// NETWORK 6
Timer3(
    BOOL_SIGNAL_IN := CollectTimerComplete OR bDirectDrainInProcess,
    BOOL_TIMER_RST := NOT bMainOnOff OR NOT bDirectDrainInProcess,
    INT_AUTO_RST := 1,
    INT_SV_SEC := iDrainingTimer); // DOWN_COUNT_TIMER
DrainComplete := Timer3.SIGNAL_BOOL;

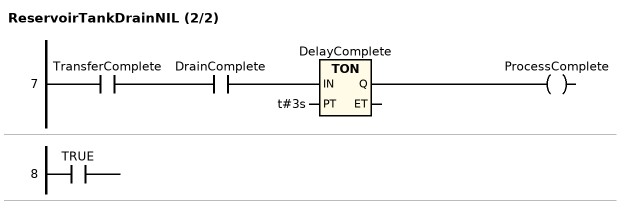
// NETWORK 7
DelayComplete(IN := TransferComplete AND DrainComplete, PT := t#3s); // TON
ProcessComplete := DelayComplete.Q;

// NETWORK 8

END_FUNCTION_BLOCK

// ---- FBs/B_JKS_NewFB/FBP-ArmRelated/fbA1_ArmHorzPosMemory.TcPOU
FUNCTION_BLOCK fbA1_ArmHorzPosMemory

VAR_INPUT PERSISTENT
	DSA1ArmHorzPosInput : DSA1_ArmHorzPosInput;
END_VAR



VAR_OUTPUT PERSISTENT
	DSA1ArmHorzPosOutput : DSA1_ArmHorzPosOutput;
END_VAR


VAR PERSISTENT

	iToleranceP: INT;

	lrBufferLdHookPosToleranceP: LREAL;
	lrBufferLdUnhookPosToleranceP: LREAL;
	lrBufferUldHookPosToleranceP: LREAL;
	lrBufferUldUnhookPosToleranceP: LREAL;

	ARlrBufferStnHookPosToleranceP: ARRAY [0..iHorzArmPosArrayQty] OF LREAL;
	ARlrBufferStnUnhookPosToleranceP: ARRAY [0..iHorzArmPosArrayQty] OF LREAL;

	iToleranceN: INT;

	lrBufferLdHookPosToleranceN: LREAL;
	lrBufferLdUnhookPosToleranceN: LREAL;
	lrBufferUldHookPosToleranceN: LREAL;
	lrBufferUldUnhookPosToleranceN: LREAL;

	ARlrBufferStnHookPosToleranceN: ARRAY [0..iHorzArmPosArrayQty] OF LREAL;
	ARlrBufferStnUnhookPosToleranceN: ARRAY [0..iHorzArmPosArrayQty] OF LREAL;

	i2ndSpdP: INT;

	lrBufferLdHookPos2ndSpdP: LREAL;
	lrBufferLdUnhookPos2ndSpdP: LREAL;
	lrBufferUldHookPos2ndSpdP: LREAL;
	lrBufferUldUnhookPos2ndSpdP: LREAL;

	ARlrBufferStnHookPos2ndSpdP: ARRAY [0..iHorzArmPosArrayQty] OF LREAL;
	ARlrBufferStnUnhookPos2ndSpdP: ARRAY [0..iHorzArmPosArrayQty] OF LREAL;

	i2ndSpdN: INT;

	lrBufferLdHookPos2ndSpdN: LREAL;
	lrBufferLdUnhookPos2ndSpdN: LREAL;
	lrBufferUldHookPos2ndSpdN: LREAL;
	lrBufferUldUnhookPos2ndSpdN: LREAL;

	ARlrBufferStnHookPos2ndSpdN: ARRAY [0..iHorzArmPosArrayQty] OF LREAL;
	ARlrBufferStnUnhookPos2ndSpdN: ARRAY [0..iHorzArmPosArrayQty] OF LREAL;
END_VAR

VAR
	iPosConfirmFL: INT;
	i2ndSpdFL: INT;
END_VAR

(* Generate Positive Tolerance *)
(*[][][][][][][][][][][][][][][][][][][][][][][][][][][][][][][][][][][][][][][][][][][][][][][][][][][][][][][][][][][][][][][][][][][][][][][][][][][][][][][][][][][][][][][][][][][][][][][][][][][]*)

lrBufferLdHookPosToleranceP := DSA1ArmHorzPosInput.lrLdHookPos + DSA1ArmHorzPosInput.lrPosConfirmToleranceSV;
lrBufferLdUnhookPosToleranceP := DSA1ArmHorzPosInput.lrLdUnhookPos + DSA1ArmHorzPosInput.lrPosConfirmToleranceSV;
lrBufferUldHookPosToleranceP := DSA1ArmHorzPosInput.lrUldHookPos + DSA1ArmHorzPosInput.lrPosConfirmToleranceSV;
lrBufferUldUnhookPosToleranceP := DSA1ArmHorzPosInput.lrUldUnhookPos + DSA1ArmHorzPosInput.lrPosConfirmToleranceSV;

iToleranceP := 1;

FOR iToleranceP := 1 TO iHorzArmPosArrayQty DO
	ARlrBufferStnHookPosToleranceP[iToleranceP] := DSA1ArmHorzPosInput.ARlrStnHookPos[iToleranceP] + DSA1ArmHorzPosInput.lrPosConfirmToleranceSV;
	ARlrBufferStnUnhookPosToleranceP[iToleranceP] := DSA1ArmHorzPosInput.ARlrStnUnhookPos[iToleranceP] + DSA1ArmHorzPosInput.lrPosConfirmToleranceSV;
END_FOR


(*[][][][][][][][][][][][][][][][][][][][][][][][][][][][][][][][][][][][][][][][][][][][][][][][][][][][][][][][][][][][][][][][][][][][][][][][][][][][][][][][][][][][][][][][][][][][][][][][][][][]*)


(* Generate Negative Tolerance *)
(*[][][][][][][][][][][][][][][][][][][][][][][][][][][][][][][][][][][][][][][][][][][][][][][][][][][][][][][][][][][][][][][][][][][][][][][][][][][][][][][][][][][][][][][][][][][][][][][][][][][]*)

lrBufferLdHookPosToleranceN := DSA1ArmHorzPosInput.lrLdHookPos - DSA1ArmHorzPosInput.lrPosConfirmToleranceSV;
lrBufferLdUnhookPosToleranceN := DSA1ArmHorzPosInput.lrLdUnhookPos - DSA1ArmHorzPosInput.lrPosConfirmToleranceSV;
lrBufferUldHookPosToleranceN := DSA1ArmHorzPosInput.lrUldHookPos - DSA1ArmHorzPosInput.lrPosConfirmToleranceSV;
lrBufferUldUnhookPosToleranceN := DSA1ArmHorzPosInput.lrUldUnhookPos - DSA1ArmHorzPosInput.lrPosConfirmToleranceSV;

iToleranceN := 1;

FOR iToleranceN := 1 TO iHorzArmPosArrayQty DO
	ARlrBufferStnHookPosToleranceN[iToleranceN] := DSA1ArmHorzPosInput.ARlrStnHookPos[iToleranceN] - DSA1ArmHorzPosInput.lrPosConfirmToleranceSV;
	ARlrBufferStnUnhookPosToleranceN[iToleranceN] := DSA1ArmHorzPosInput.ARlrStnUnhookPos[iToleranceN] - DSA1ArmHorzPosInput.lrPosConfirmToleranceSV;
END_FOR


(*[][][][][][][][][][][][][][][][][][][][][][][][][][][][][][][][][][][][][][][][][][][][][][][][][][][][][][][][][][][][][][][][][][][][][][][][][][][][][][][][][][][][][][][][][][][][][][][][][][][]*)



(* Generate Positive 2ndSpeed *)
(*[][][][][][][][][][][][][][][][][][][][][][][][][][][][][][][][][][][][][][][][][][][][][][][][][][][][][][][][][][][][][][][][][][][][][][][][][][][][][][][][][][][][][][][][][][][][][][][][][][][]*)

lrBufferLdHookPos2ndSpdP := DSA1ArmHorzPosInput.lrLdHookPos + DSA1ArmHorzPosInput.lr2ndSpeedSV;
lrBufferLdUnhookPos2ndSpdP := DSA1ArmHorzPosInput.lrLdUnhookPos + DSA1ArmHorzPosInput.lr2ndSpeedSV;
lrBufferUldHookPos2ndSpdP := DSA1ArmHorzPosInput.lrUldHookPos + DSA1ArmHorzPosInput.lr2ndSpeedSV;
lrBufferUldUnhookPos2ndSpdP := DSA1ArmHorzPosInput.lrUldUnhookPos + DSA1ArmHorzPosInput.lr2ndSpeedSV;

i2ndSpdP := 1;

FOR i2ndSpdP := 1 TO iHorzArmPosArrayQty DO
	ARlrBufferStnHookPos2ndSpdP[i2ndSpdP] := DSA1ArmHorzPosInput.ARlrStnHookPos[i2ndSpdP] + DSA1ArmHorzPosInput.lr2ndSpeedSV;
	ARlrBufferStnUnhookPos2ndSpdP[i2ndSpdP] := DSA1ArmHorzPosInput.ARlrStnUnhookPos[i2ndSpdP] + DSA1ArmHorzPosInput.lr2ndSpeedSV;
END_FOR


(*[][][][][][][][][][][][][][][][][][][][][][][][][][][][][][][][][][][][][][][][][][][][][][][][][][][][][][][][][][][][][][][][][][][][][][][][][][][][][][][][][][][][][][][][][][][][][][][][][][][]*)


(* Generate Negative 2ndSpeed *)
(*[][][][][][][][][][][][][][][][][][][][][][][][][][][][][][][][][][][][][][][][][][][][][][][][][][][][][][][][][][][][][][][][][][][][][][][][][][][][][][][][][][][][][][][][][][][][][][][][][][][]*)

lrBufferLdHookPos2ndSpdN := DSA1ArmHorzPosInput.lrLdHookPos - DSA1ArmHorzPosInput.lr2ndSpeedSV;
lrBufferLdUnhookPos2ndSpdN := DSA1ArmHorzPosInput.lrLdUnhookPos - DSA1ArmHorzPosInput.lr2ndSpeedSV;
lrBufferUldHookPos2ndSpdN := DSA1ArmHorzPosInput.lrUldHookPos - DSA1ArmHorzPosInput.lr2ndSpeedSV;
lrBufferUldUnhookPos2ndSpdN := DSA1ArmHorzPosInput.lrUldUnhookPos - DSA1ArmHorzPosInput.lr2ndSpeedSV;

i2ndSpdN := 1;

FOR i2ndSpdN := 1 TO iHorzArmPosArrayQty DO
	ARlrBufferStnHookPos2ndSpdN[i2ndSpdN] := DSA1ArmHorzPosInput.ARlrStnHookPos[i2ndSpdN] - DSA1ArmHorzPosInput.lr2ndSpeedSV;
	ARlrBufferStnUnhookPos2ndSpdN[i2ndSpdN] := DSA1ArmHorzPosInput.ARlrStnUnhookPos[i2ndSpdN] - DSA1ArmHorzPosInput.lr2ndSpeedSV;
END_FOR


(*[][][][][][][][][][][][][][][][][][][][][][][][][][][][][][][][][][][][][][][][][][][][][][][][][][][][][][][][][][][][][][][][][][][][][][][][][][][][][][][][][][][][][][][][][][][][][][][][][][][]*)


(*Generate Pos Confirm Bit*)
(*[][][][][][][][][][][][][][][][][][][][][][][][][][][][][][][][][][][][][][][][][][][][][][][][][][][][][][][][][][][][][][][][][][][][][][][][][][][][][][][][][][][][][][][][][][][][][][][][][][][]*)
IF DSA1ArmHorzPosInput.lrCurrentPos >= lrBufferLdHookPosToleranceN  AND DSA1ArmHorzPosInput.lrCurrentPos <= lrBufferLdHookPosToleranceP THEN
DSA1ArmHorzPosOutput.bLdHookPosConfirm := TRUE;
ELSE
DSA1ArmHorzPosOutput.bLdHookPosConfirm := FALSE;
END_IF

IF DSA1ArmHorzPosInput.lrCurrentPos >= lrBufferLdUnhookPosToleranceN  AND DSA1ArmHorzPosInput.lrCurrentPos <= lrBufferLdUnhookPosToleranceP THEN
DSA1ArmHorzPosOutput.bLdUnhookPosConfirm := TRUE;
ELSE
DSA1ArmHorzPosOutput.bLdUnhookPosConfirm := FALSE;
END_IF

IF DSA1ArmHorzPosInput.lrCurrentPos >= lrBufferUldHookPosToleranceN  AND DSA1ArmHorzPosInput.lrCurrentPos <= lrBufferUldHookPosToleranceP THEN
DSA1ArmHorzPosOutput.bUldHookPosConfirm := TRUE;
ELSE
DSA1ArmHorzPosOutput.bUldHookPosConfirm := FALSE;
END_IF

IF DSA1ArmHorzPosInput.lrCurrentPos >= lrBufferUldUnhookPosToleranceN  AND DSA1ArmHorzPosInput.lrCurrentPos <= lrBufferUldUnhookPosToleranceP THEN
DSA1ArmHorzPosOutput.bUldUnhookPosConfirm := TRUE;
ELSE
DSA1ArmHorzPosOutput.bUldUnhookPosConfirm := FALSE;
END_IF


iPosConfirmFL := 1;
FOR iPosConfirmFL := 1 TO iHorzArmPosArrayQty DO

		IF DSA1ArmHorzPosInput.lrCurrentPos >= ARlrBufferStnHookPosToleranceN[iPosConfirmFL]  AND DSA1ArmHorzPosInput.lrCurrentPos <= ARlrBufferStnHookPosToleranceP[iPosConfirmFL] THEN
		DSA1ArmHorzPosOutput.ARbStnHookPosConfirm[iPosConfirmFL] := TRUE;
		ELSE
		DSA1ArmHorzPosOutput.ARbStnHookPosConfirm[iPosConfirmFL] := FALSE;
		END_IF

		IF DSA1ArmHorzPosInput.lrCurrentPos >= ARlrBufferStnUnhookPosToleranceN[iPosConfirmFL]  AND DSA1ArmHorzPosInput.lrCurrentPos <= ARlrBufferStnUnhookPosToleranceP[iPosConfirmFL] THEN
		DSA1ArmHorzPosOutput.ARbStnUnhookPosConfirm[iPosConfirmFL] := TRUE;
		ELSE
		DSA1ArmHorzPosOutput.ARbStnUnhookPosConfirm[iPosConfirmFL] := FALSE;
		END_IF

END_FOR

(*[][][][][][][][][][][][][][][][][][][][][][][][][][][][][][][][][][][][][][][][][][][][][][][][][][][][][][][][][][][][][][][][][][][][][][][][][][][][][][][][][][][][][][][][][][][][][][][][][][][]*)



(*Generate 2nd Speed Bit*)
(*[][][][][][][][][][][][][][][][][][][][][][][][][][][][][][][][][][][][][][][][][][][][][][][][][][][][][][][][][][][][][][][][][][][][][][][][][][][][][][][][][][][][][][][][][][][][][][][][][][][]*)
IF DSA1ArmHorzPosInput.lrCurrentPos >= lrBufferLdHookPos2ndSpdN  AND DSA1ArmHorzPosInput.lrCurrentPos <= lrBufferLdHookPos2ndSpdP AND DSA1ArmHorzPosInput.lrTargetPos = DSA1ArmHorzPosInput.lrLdHookPos THEN


DSA1ArmHorzPosOutput.bLdHook2ndSpeedEn := TRUE;
ELSE
DSA1ArmHorzPosOutput.bLdHook2ndSpeedEn := FALSE;
END_IF

IF DSA1ArmHorzPosInput.lrCurrentPos >= lrBufferLdUnhookPos2ndSpdN  AND DSA1ArmHorzPosInput.lrCurrentPos <= lrBufferLdUnhookPos2ndSpdP AND DSA1ArmHorzPosInput.lrTargetPos = DSA1ArmHorzPosInput.lrLdUnhookPos THEN
DSA1ArmHorzPosOutput.bLdUnhook2ndSpeedEn := TRUE;
ELSE
DSA1ArmHorzPosOutput.bLdUnhook2ndSpeedEn := FALSE;
END_IF

IF DSA1ArmHorzPosInput.lrCurrentPos >= lrBufferUldHookPos2ndSpdN  AND DSA1ArmHorzPosInput.lrCurrentPos <= lrBufferUldHookPos2ndSpdP AND DSA1ArmHorzPosInput.lrTargetPos = DSA1ArmHorzPosInput.lrUldHookPos THEN
DSA1ArmHorzPosOutput.bUldHook2ndSpeedEn := TRUE;
ELSE
DSA1ArmHorzPosOutput.bUldHook2ndSpeedEn := FALSE;
END_IF

IF DSA1ArmHorzPosInput.lrCurrentPos >= lrBufferUldUnhookPos2ndSpdN  AND DSA1ArmHorzPosInput.lrCurrentPos <= lrBufferUldUnhookPos2ndSpdP AND DSA1ArmHorzPosInput.lrTargetPos = DSA1ArmHorzPosInput.lrUldUnhookPos THEN
DSA1ArmHorzPosOutput.bUldUnhook2ndSpeedEn := TRUE;
ELSE
DSA1ArmHorzPosOutput.bUldUnhook2ndSpeedEn := FALSE;
END_IF


i2ndSpdFL := 1;
FOR i2ndSpdFL := 1 TO iHorzArmPosArrayQty DO

	IF DSA1ArmHorzPosInput.lrCurrentPos >= ARlrBufferStnHookPos2ndSpdN[i2ndSpdFL]  AND DSA1ArmHorzPosInput.lrCurrentPos <= ARlrBufferStnHookPos2ndSpdP[i2ndSpdFL] AND DSA1ArmHorzPosInput.lrTargetPos = DSA1ArmHorzPosInput.ARlrStnHookPos[i2ndSpdFL] THEN
	DSA1ArmHorzPosOutput.ARbStnHook2ndSpeedEn[i2ndSpdFL] := TRUE;
	ELSE
	DSA1ArmHorzPosOutput.ARbStnHook2ndSpeedEn[i2ndSpdFL] := FALSE;
	END_IF

	IF DSA1ArmHorzPosInput.lrCurrentPos >= ARlrBufferStnUnhookPos2ndSpdN[i2ndSpdFL]  AND DSA1ArmHorzPosInput.lrCurrentPos <= ARlrBufferStnUnhookPos2ndSpdP[i2ndSpdFL] AND DSA1ArmHorzPosInput.lrTargetPos = DSA1ArmHorzPosInput.ARlrStnUnhookPos[i2ndSpdFL] THEN
	DSA1ArmHorzPosOutput.ARbStnUnhook2ndSpeedEn[i2ndSpdFL] := TRUE;
	ELSE
	DSA1ArmHorzPosOutput.ARbStnUnhook2ndSpeedEn[i2ndSpdFL] := FALSE;
	END_IF

END_FOR

(*[][][][][][][][][][][][][][][][][][][][][][][][][][][][][][][][][][][][][][][][][][][][][][][][][][][][][][][][][][][][][][][][][][][][][][][][][][][][][][][][][][][][][][][][][][][][][][][][][][][]*)




(*
IN

	DSA1ArmHorzPosInput.lrTargetPos

	DSA1ArmHorzPosInput.lrPosConfirmToleranceSV
	DSA1ArmHorzPosInput.lr2ndSpeedSV

	DSA1ArmHorzPosInput.lrLdHookPos
	DSA1ArmHorzPosInput.lrLdUnhookPos

	DSA1ArmHorzPosInput.lrUldHookPos 
	DSA1ArmHorzPosInput.lrUldUnhookPos

	DSA1ArmHorzPosInput.ARlrStnHookPos
	DSA1ArmHorzPosInput.ARlrStnUnhookPos


OUT

	DSA1ArmHorzPosOutput.bLdHookPosConfirm
	DSA1ArmHorzPosOutput.bLdUnhookPosConfirm
	DSA1ArmHorzPosOutput.bUldHookPosConfirm
	DSA1ArmHorzPosOutput.bUldUnhookPosConfirm
	DSA1ArmHorzPosOutput.ARbStnHookPosConfirm
	DSA1ArmHorzPosOutput.ARbStnUnhookPosConfirm

	DSA1ArmHorzPosOutput.bLdHook2ndSpeedEn
	DSA1ArmHorzPosOutput.bLdUnhook2ndSpeedEn 
	DSA1ArmHorzPosOutput.bUldHook2ndSpeedEn
	DSA1ArmHorzPosOutput.bUldUnhook2ndSpeedEn 
	DSA1ArmHorzPosOutput.ARbStnHook2ndSpeedEn
	DSA1ArmHorzPosOutput.ARbStnUnhook2ndSpeedEn
*)

END_FUNCTION_BLOCK

// ---- FBs/B_JKS_NewFB/FBP-ArmRelated/fbFBPArmHorzZoneConfirm.TcPOU
FUNCTION_BLOCK fbFBPArmHorzZoneConfirm
VAR_INPUT
	bEnable 					: BOOL;
(*	iLdStnID					: INT;
	iUldStnID					: INT;
*)	lrHorzActualPos 			: LREAL;
	lrHorzStartPoint 			: LREAL;
	lrHorzEndPoint 			: LREAL;
	lrLdHorzCentrePoint 		: LREAL;
	ARlrStnHorzCentrePoint 	: ARRAY [1..iStnQty] OF LREAL;
	lrUldHorzCentrePoint 		: LREAL;
	ARiStnHorzListing 		: ARRAY [1..50] OF INT;

END_VAR


VAR_OUTPUT
	bLdHorzZoneConfirm 		: BOOL;
	ARbHorzStnZoneConfirm 	: ARRAY [1..iStnQty] OF BOOL;
	bUldHorzZoneConfirm 		: BOOL;
	ICurrentHorzZoneNo 			: INT;
	bInvalidListingErr				: BOOL;



END_VAR
(*
VAR_IN_OUT
	iZoneEndPoint : ARRAY [1..20] OF INT;
	iActualPos: INT;

END_VAR
*)
VAR

	iActualPos: INT;


	bEnableRE: R_TRIG;
	iGenZoneFL: INT;
	ARlrZoneCentrePoint : ARRAY [1..50] OF LREAL;
	ARlrZoneEndPoint : ARRAY [1..50] OF LREAL;
	ARbZonePosConfirmInt : ARRAY [1..50] OF BOOL;
	iCheckListFL: INT;
	iEndPointFL: INT;
	bEnableFE: F_TRIG;
	iClearFL: INT;
	IZonePosCfFL: INT;
	iCurrentStnFL: INT;
	bCheckStnConfirm: BOOL;
	iCheckStnBitFL: INT;
END_VAR

(*bEnable Rising Edge*)
bEnableRE(CLK:=bEnable , Q=> );
bEnableFE(CLK:=bEnable , Q=> );

(*Generate Zone Centre Point and Transfer Confirm Bit*)
IF bEnable THEN
iGenZoneFL := 1;
	FOR iGenZoneFL := 1 TO 50 DO
		IF iGenZoneFL >= 1 AND iGenZoneFL <= 50 THEN

			IF ARiStnHorzListing[iGenZoneFL] = iLdStnID THEN
				ARlrZoneCentrePoint[iGenZoneFL] := lrLdHorzCentrePoint;
				bLdHorzZoneConfirm := ARbZonePosConfirmInt[iGenZoneFL];
			END_IF

			IF ARiStnHorzListing[iGenZoneFL] = iUldStnID THEN
				ARlrZoneCentrePoint[iGenZoneFL] := lrUldHorzCentrePoint;
				bUldHorzZoneConfirm := ARbZonePosConfirmInt[iGenZoneFL];
			END_IF

			IF ARiStnHorzListing[iGenZoneFL] <> iUldStnID AND ARiStnHorzListing[iGenZoneFL] <> iUldStnID AND ARiStnHorzListing[iGenZoneFL] <> 0 AND ARiStnHorzListing[iGenZoneFL] <= iStnQty THEN
				ARlrZoneCentrePoint[iGenZoneFL] := ARlrStnHorzCentrePoint[ARiStnHorzListing[iGenZoneFL]];
				ARbHorzStnZoneConfirm[ARiStnHorzListing[iGenZoneFL]] := ARbZonePosConfirmInt[iGenZoneFL];
			END_IF
		END_IF
	END_FOR
END_IF


(*Check invalid Stn Listing*)
IF bEnableRE.Q THEN
bInvalidListingErr := FALSE;
iCheckListFL := 1;
	FOR iCheckListFL := 1 TO 50 DO
		IF iCheckListFL >= 1 AND iCheckListFL <= 50 THEN

			IF iCheckListFL = 1 AND ARlrZoneCentrePoint[1] <= 0 THEN
			bInvalidListingErr := TRUE;
			iCheckListFL := 50+1;
			END_IF

			IF iCheckListFL > 1 AND ARlrZoneCentrePoint[iCheckListFL] <= ARlrZoneCentrePoint[iCheckListFL-1] AND ARiStnHorzListing[iCheckListFL] >0 THEN
			bInvalidListingErr := TRUE;
			iCheckListFL := 50+1;
			END_IF
		END_IF
	END_FOR
END_IF




(*Generate End Point *)
IF bEnableRE.Q THEN
iEndPointFL := 1;
	FOR iEndPointFL := 1 TO 50 DO
		IF iEndPointFL >= 1 AND iEndPointFL <= 50-1 THEN

(*			IF iEndPointFL >1 THEN*)
				IF ((ARlrZoneCentrePoint[iEndPointFL+1] - ARlrZoneCentrePoint[iEndPointFL])/2) >0 THEN
				ARlrZoneEndPoint[iEndPointFL] := ((ARlrZoneCentrePoint[iEndPointFL+1] - ARlrZoneCentrePoint[iEndPointFL])/2)+ARlrZoneCentrePoint[iEndPointFL];
				ELSIF lrHorzEndPoint <= ARlrZoneCentrePoint[iEndPointFL] THEN
				ARlrZoneEndPoint[iEndPointFL] := ARlrZoneCentrePoint[iEndPointFL]+5000;
				iEndPointFL := 50+1;
				ELSIF lrHorzEndPoint > ARlrZoneCentrePoint[iEndPointFL] THEN
				ARlrZoneEndPoint[iEndPointFL] := lrHorzEndPoint+1;
				iEndPointFL := 50+1;
				END_IF
(*			END_IF*)
		END_IF
	END_FOR
END_IF


(*Clear Data*)
IF bEnableFE.Q THEN
iClearFL := 1;
	FOR iClearFL := 1 TO 50 DO
		IF iClearFL >= 1 AND iClearFL <= 50 THEN

			ARlrZoneCentrePoint[iClearFL] := 0;
			ARlrZoneEndPoint[iClearFL] := 0;
			ARbZonePosConfirmInt[iClearFL] := FALSE;

			IF iClearFL >= 1 AND iClearFL <= iStnQty THEN
			ARbHorzStnZoneConfirm[iClearFL] := FALSE;
			END_IF

		END_IF
	END_FOR
bLdHorzZoneConfirm := FALSE;
bUldHorzZoneConfirm := FALSE;
ICurrentHorzZoneNo := 0;
bInvalidListingErr := FALSE;
END_IF


(*Convert LREAL to INT*)


iActualPos := LREAL_TO_INT(lrHorzActualPos);




IF bEnable AND NOT bInvalidListingErr THEN


(*General Zone Pos Confirm Internal*)
IZonePosCfFL := 1;
	FOR IZonePosCfFL := 1 TO 50 DO
		IF IZonePosCfFL >= 1 AND IZonePosCfFL <= 50 THEN

			IF IZonePosCfFL = 1 THEN
				IF (iActualPos >= lrHorzStartPoint) AND (iActualPos < ARlrZoneEndPoint[IZonePosCfFL]) AND iActualPos >0 THEN
				ARbZonePosConfirmInt[IZonePosCfFL] := TRUE;
				ELSE
				ARbZonePosConfirmInt[IZonePosCfFL] := FALSE;
				END_IF
			END_IF

			IF IZonePosCfFL > 1 THEN
				IF (iActualPos >= ARlrZoneEndPoint[IZonePosCfFL-1]) AND (iActualPos < ARlrZoneEndPoint[IZonePosCfFL]) AND iActualPos >0 THEN
				ARbZonePosConfirmInt[IZonePosCfFL] := TRUE;
				ELSE
				ARbZonePosConfirmInt[IZonePosCfFL] := FALSE;
				END_IF
			END_IF
		END_IF
	END_FOR

(*Generate ICurrentHorzZoneNo *)


	IF bLdHorzZoneConfirm THEN
	ICurrentHorzZoneNo := iLdStnID;
	ELSIF bUldHorzZoneConfirm THEN
	ICurrentHorzZoneNo := iUldStnID;
	ELSE
	iCurrentStnFL := 1;
	
		FOR iCurrentStnFL := 1 TO iStnQty DO
			IF iCurrentStnFL >= 1 AND iCurrentStnFL <= iStnQty THEN

				IF ARbHorzStnZoneConfirm[iCurrentStnFL] THEN
				ICurrentHorzZoneNo := iCurrentStnFL;
				END_IF
	
			END_IF
		END_FOR
	
	END_IF

(*Check if any Ld/Uld/Stn Pos Confirm Bit is on, else -> ICurrentHorzZoneNo := 0; *)
bCheckStnConfirm := FALSE;
iCheckStnBitFL := 1;

	FOR iCheckStnBitFL := 1 TO iStnQty DO
		IF iCheckStnBitFL >= 1 AND iCheckStnBitFL <= iStnQty THEN
			IF ARbHorzStnZoneConfirm[iCheckStnBitFL] THEN
			bCheckStnConfirm := TRUE;
			END_IF
		END_IF
	END_FOR


	IF NOT bLdHorzZoneConfirm AND NOT bUldHorzZoneConfirm AND NOT bCheckStnConfirm THEN
	ICurrentHorzZoneNo := 0;
	END_IF

END_IF

END_FUNCTION_BLOCK

// ---- FBs/B_JKS_NewFB/FBP-ArmRelated/fbFBPVertArmPosConfirm.TcPOU
FUNCTION_BLOCK fbFBPVertArmPosConfirm
VAR_INPUT
	bEnable 						: BOOL;
(*	iLdStnID						: INT;
	iUldStnID						: INT;
*)	lrCurrentVertActualPos 		: LREAL; (*From Encoder Reading*)
	iCurrentHorzZoneNo 			: INT; (*From fbFBPArmZoneConfirm Output*)
	DSLdZonePosOut 			: DSA32_StationZonePosOut; (*From fbGnrProductRecipeMemory Output*)
	ARDSStationZonePosOut 	: ARRAY [0..iStnQty] OF DSA32_StationZonePosOut; (*From fbGnrProductRecipeMemory Output*)
	DSUldZonePosOut 			: DSA32_StationZonePosOut; (*From fbGnrProductRecipeMemory Output*)



END_VAR
VAR_OUTPUT
	bVertTopTravelPosConfirm 	: BOOL;
	bVertMidTravelPosConfirm 	: BOOL;
	bVertDownPosConfirm 		: BOOL;


END_VAR
VAR
	DSBufferZonePosOut : DSA32_StationZonePosOut;
	DSEmptyZonePosOut : DSA32_StationZonePosOut;
	iBufferFL: INT;
END_VAR

(*Pos Confirm Checking Start*)
IF bEnable THEN

	(*Find Station DS and Push to buffer*)
	IF iCurrentHorzZoneNo = iLdStnID THEN
		DSBufferZonePosOut := DSLdZonePosOut;
	ELSIF iCurrentHorzZoneNo = iUldStnID THEN
		DSBufferZonePosOut := DSUldZonePosOut;
	ELSIF iCurrentHorzZoneNo > 0 THEN
		iBufferFL := 1;
			FOR iBufferFL := 1 TO iStnQty DO
				IF iBufferFL >= 1 AND iBufferFL <= iStnQty THEN
					IF iCurrentHorzZoneNo = iBufferFL THEN
					DSBufferZonePosOut := ARDSStationZonePosOut[iBufferFL];
					END_IF
				END_IF
			END_FOR
	ELSE
		DSBufferZonePosOut := DSEmptyZonePosOut;
	END_IF

(*Generate Bit*)

	IF DSBufferZonePosOut.lrZone1StartPos > 1 AND DSBufferZonePosOut.lrZone1StartPos = lrCurrentVertActualPos THEN
	bVertTopTravelPosConfirm := TRUE;
	ELSE
	bVertTopTravelPosConfirm := FALSE;
	END_IF

	IF DSBufferZonePosOut.lrMidPos > 1 AND DSBufferZonePosOut.lrMidPos = lrCurrentVertActualPos THEN
	bVertMidTravelPosConfirm := TRUE;
	ELSE
	bVertMidTravelPosConfirm := FALSE;
	END_IF

	IF DSBufferZonePosOut.lrZone4EndPos > 1 AND DSBufferZonePosOut.lrZone4EndPos = lrCurrentVertActualPos THEN
	bVertDownPosConfirm := TRUE;
	ELSE
	bVertDownPosConfirm := FALSE;
	END_IF




END_IF





(*Reset*)
IF NOT bEnable OR iCurrentHorzZoneNo <= 0 THEN
	bVertTopTravelPosConfirm 	:= FALSE;
	bVertMidTravelPosConfirm 	:= FALSE;
	bVertDownPosConfirm 		:= FALSE;
	DSBufferZonePosOut := DSEmptyZonePosOut;

END_IF

END_FUNCTION_BLOCK

// ---- FBs/B_JKS_NewFB/FBP-EncoderIncrementalCtrl/fbEncoderConversion.TcPOU
FUNCTION_BLOCK fbEncoderConversion
VAR_INPUT
	bCounterValueReset 				: BOOL;
	bIN_SetCounterDone 				: BOOL;
	udIN_CounterValue 				: UDINT;
	bInvertCounterValueEn				: BOOL;
	bCounterValueErrReset			: BOOL;
END_VAR
VAR_OUTPUT
	bOUT_SetCounterEn 				: BOOL;
	udOUT_SetCounterValue 			: UDINT;
	lrPositionMM 						: LREAL;
	bCounterValueErr					: BOOL;
END_VAR

VAR_IN_OUT PERSISTENT
	lrRatioPulseToMM 				: LREAL;
	iCounterValueResetTime_Sec 		: INT;

END_VAR

VAR
	bCounterValueResetRE			: R_TRIG;
	tCounterValueReset				: TON;
	bCounterValueResetHR			: BOOL;
	tCounterValueResetOnTime		: TON;
	tCounterValueResetTimeout: TON;
	diInternalCounterValue: DINT;
END_VAR

(*Set Minimum Control*)
IF iCounterValueResetTime_Sec < 2 THEN
iCounterValueResetTime_Sec := 2;
END_IF

IF lrRatioPulseToMM < 1 THEN
lrRatioPulseToMM := 1;
END_IF


(*Preparation*)
bCounterValueResetRE(CLK:= bCounterValueReset, Q=> );

IF bCounterValueResetRE.Q AND NOT bCounterValueErr THEN
bCounterValueResetHR := TRUE;
END_IF

tCounterValueResetOnTime(IN:= bCounterValueResetHR, PT:=t#1s , Q=> , ET=> );

(*Counter Reset Start*)
IF bCounterValueResetHR AND NOT tCounterValueResetOnTime.Q THEN
bOUT_SetCounterEn := TRUE;
ELSE
bOUT_SetCounterEn := FALSE;
END_IF

(*Counter Reset Completed Flag*)
IF bIN_SetCounterDone THEN
bCounterValueResetHR := FALSE;
END_IF

(*Check If Counter not able to reset*)
tCounterValueResetTimeout(IN:=bCounterValueResetHR , PT:=INT_TO_TIME(iCounterValueResetTime_Sec*1000) , Q=> , ET=> );

IF tCounterValueResetTimeout.Q THEN
bCounterValueErr := TRUE;
END_IF

(*ResetError*)
IF bCounterValueErrReset THEN
bCounterValueErr := FALSE;
END_IF


(*Value Convert To Counter with LREAL*)
(**********************
0		= -2147483647
2147483648 	= 0 , 
4294967295 	= +2147483647
***********************)

udOUT_SetCounterValue := 2147483648;

IF NOT bInvertCounterValueEn THEN
diInternalCounterValue := udIN_CounterValue - 2147483648;
ELSE
diInternalCounterValue :=  2147483648 - udIN_CounterValue;
END_IF

lrPositionMM := DINT_TO_LREAL(diInternalCounterValue) / lrRatioPulseToMM;

END_FUNCTION_BLOCK

// ---- FBs/B_JKS_NewFB/FBP-HMIAddMapping/fbHMIAddMappingArrayBool.TcPOU
FUNCTION_BLOCK fbHMIAddMappingArrayBool


VAR_INPUT
	bEN : BOOL;
END_VAR

VAR_IN_OUT PERSISTENT
	ARbBoolAddress_Pro 					: ARRAY [0..iAddMapArrayBool] OF BOOL;
	ARbBoolAddress_Hmi 				: ARRAY [0..iAddMapArrayBool] OF BOOL;
END_VAR


VAR_OUTPUT
END_VAR


VAR
	ARBufferbBoolAddress_Pro 				:  ARRAY [1..iAddMapArrayBool] OF BOOL;
	ARBufferbBoolAddress_Hmi 				:  ARRAY [1..iAddMapArrayBool] OF BOOL;

	ARUpdate_bBoolAddress_Pro 				:  ARRAY [1..iAddMapArrayBool] OF BOOL;
	ARUpdate_bBoolAddress_Hmi 				:  ARRAY [1..iAddMapArrayBool] OF BOOL;

	iInitialFL: INT;
	iProgramFL: INT;
	bENRE : R_TRIG;


END_VAR

(*Initialized*)
bENRE(CLK:=bEN , Q=> );
IF bENRE.Q THEN
			(*Bool*)
iInitialFL := 1;

	FOR iInitialFL := 1 TO iAddMapArrayBool DO
			ARBufferbBoolAddress_Pro[iInitialFL] := ARbBoolAddress_Pro[iInitialFL];
			ARBufferbBoolAddress_Hmi[iInitialFL] := ARbBoolAddress_Pro[iInitialFL];
			ARbBoolAddress_Hmi[iInitialFL] := ARbBoolAddress_Pro[iInitialFL];
	END_FOR

END_IF

(*Program*)

			(**********PRO Side Value Change**********)

iProgramFL:= 1;

	FOR iProgramFL := 1 TO iAddMapArrayBool DO

		ARUpdate_bBoolAddress_Pro[iProgramFL] := FALSE;

			IF ARBufferbBoolAddress_Pro[iProgramFL] <> ARbBoolAddress_Pro[iProgramFL] THEN
				ARUpdate_bBoolAddress_Pro[iProgramFL] := TRUE;
			END_IF
		
			IF ARUpdate_bBoolAddress_Pro[iProgramFL] THEN
				ARBufferbBoolAddress_Pro[iProgramFL] := ARbBoolAddress_Pro[iProgramFL];
				ARBufferbBoolAddress_Hmi[iProgramFL] := ARbBoolAddress_Pro[iProgramFL];
				ARbBoolAddress_Hmi[iProgramFL] := ARbBoolAddress_Pro[iProgramFL];
			END_IF
		


					(**********HMI Side Value Change**********)
		
		ARUpdate_bBoolAddress_Hmi[iProgramFL] := FALSE;
		
			IF ARBufferbBoolAddress_Hmi[iProgramFL] <> ARbBoolAddress_Hmi[iProgramFL] THEN
				ARUpdate_bBoolAddress_Hmi[iProgramFL] := TRUE;
			END_IF
		
			IF ARUpdate_bBoolAddress_Hmi[iProgramFL] THEN
				ARBufferbBoolAddress_Pro[iProgramFL] := ARbBoolAddress_Hmi[iProgramFL];
				ARBufferbBoolAddress_Hmi[iProgramFL] := ARbBoolAddress_Hmi[iProgramFL];
				ARbBoolAddress_Pro[iProgramFL] := ARbBoolAddress_Hmi[iProgramFL];
			END_IF

	END_FOR
(*
(*Bool 001*)
IF NOT ARUpdate_bBoolAddress_Hmi THEN ARbBoolAddress_Pro := Pro_bBool_001; ELSE Pro_bBool_001 := ARbBoolAddress_Pro; END_IF
IF NOT ARUpdate_bBoolAddress_Pro THEN ARbBoolAddress_Hmi := Hmi_bBool_001; ELSE Hmi_bBool_001 := ARbBoolAddress_Hmi; END_IF
*)

END_FUNCTION_BLOCK

// ---- FBs/B_JKS_NewFB/FBP-HMIAddMapping/fbHMIAddMappingArrayInt.TcPOU
FUNCTION_BLOCK fbHMIAddMappingArrayInt


VAR_INPUT
	bEN : BOOL;
END_VAR

VAR_IN_OUT PERSISTENT
	ARiIntAddress_Pro 					: ARRAY [0..iAddMapArrayInt] OF INT;
	ARiIntAddress_Hmi 				: ARRAY [0..iAddMapArrayInt] OF INT;
END_VAR


VAR_OUTPUT
END_VAR


VAR
	ARBufferiIntAddress_Pro 				:  ARRAY [1..iAddMapArrayInt] OF INT;
	ARBufferiIntAddress_Hmi 				:  ARRAY [1..iAddMapArrayInt] OF INT;

	ARUpdate_bIntAddress_Pro 				:  ARRAY [1..iAddMapArrayInt] OF BOOL;
	ARUpdate_bIntAddress_Hmi 				:  ARRAY [1..iAddMapArrayInt] OF BOOL;

	iInitialFL: INT;
	iProgramFL: INT;
	bENRE : R_TRIG;


END_VAR

(*Initialized*)
bENRE(CLK:=bEN , Q=> );
IF bENRE.Q THEN
			(*Int*)
iInitialFL := 1;

	FOR iInitialFL := 1 TO iAddMapArrayInt DO
			ARBufferiIntAddress_Pro[iInitialFL] := ARiIntAddress_Pro[iInitialFL];
			ARBufferiIntAddress_Hmi[iInitialFL] := ARiIntAddress_Pro[iInitialFL];
			ARiIntAddress_Hmi[iInitialFL] := ARiIntAddress_Pro[iInitialFL];
	END_FOR

END_IF

(*Program*)

			(**********PRO Side Value Change**********)

iProgramFL:= 1;

	FOR iProgramFL := 1 TO iAddMapArrayInt DO

		ARUpdate_bIntAddress_Pro[iProgramFL] := FALSE;
		
			IF ARBufferiIntAddress_Pro[iProgramFL] <> ARiIntAddress_Pro[iProgramFL] THEN
				ARUpdate_bIntAddress_Pro[iProgramFL] := TRUE;
			END_IF

			IF ARUpdate_bIntAddress_Pro[iProgramFL] THEN
				ARBufferiIntAddress_Pro[iProgramFL] := ARiIntAddress_Pro[iProgramFL];
				ARBufferiIntAddress_Hmi[iProgramFL] := ARiIntAddress_Pro[iProgramFL];
				ARiIntAddress_Hmi[iProgramFL] := ARiIntAddress_Pro[iProgramFL];
			END_IF
		


					(**********HMI Side Value Change**********)
		
		ARUpdate_bIntAddress_Hmi[iProgramFL] := FALSE;

			IF ARBufferiIntAddress_Hmi[iProgramFL] <> ARiIntAddress_Hmi[iProgramFL] THEN
				ARUpdate_bIntAddress_Hmi[iProgramFL] := TRUE;
			END_IF
		
			IF ARUpdate_bIntAddress_Hmi[iProgramFL] THEN
				ARBufferiIntAddress_Pro[iProgramFL] := ARiIntAddress_Hmi[iProgramFL];
				ARBufferiIntAddress_Hmi[iProgramFL] := ARiIntAddress_Hmi[iProgramFL];
				ARiIntAddress_Pro[iProgramFL] := ARiIntAddress_Hmi[iProgramFL];
			END_IF

	END_FOR
(*
(*Int 001*)
IF NOT ARUpdate_bIntAddress_Hmi THEN ARiIntAddress_Pro := Pro_iInt_001; ELSE Pro_iInt_001 := ARiIntAddress_Pro; END_IF
IF NOT ARUpdate_bIntAddress_Pro THEN ARiIntAddress_Hmi := Hmi_iInt_001; ELSE Hmi_iInt_001 := ARiIntAddress_Hmi; END_IF
*)

END_FUNCTION_BLOCK

// ---- FBs/B_JKS_NewFB/FBP-HMIAddMapping/fbHMIAddMappingArrayLreal.TcPOU
FUNCTION_BLOCK fbHMIAddMappingArrayLreal


VAR_INPUT
	bEN : BOOL;
END_VAR

VAR_IN_OUT PERSISTENT
	ARlrLrealAddress_Pro 					: ARRAY [0..iAddMapArrayLreal] OF LREAL;
	ARlrLrealAddress_Hmi 				: ARRAY [0..iAddMapArrayLreal] OF LREAL;
END_VAR


VAR_OUTPUT
END_VAR


VAR
	ARBufferlrLrealAddress_Pro 				:  ARRAY [1..iAddMapArrayLreal] OF LREAL;
	ARBufferlrLrealAddress_Hmi 				:  ARRAY [1..iAddMapArrayLreal] OF LREAL;

	ARUpdate_bLrealAddress_Pro 				:  ARRAY [1..iAddMapArrayLreal] OF BOOL;
	ARUpdate_bLrealAddress_Hmi 				:  ARRAY [1..iAddMapArrayLreal] OF BOOL;

	iInitialFL: INT;
	iProgramFL: INT;
	bENRE : R_TRIG;


END_VAR

(*Initialized*)
bENRE(CLK:=bEN , Q=> );
IF bENRE.Q THEN
			(*Lreal*)
iInitialFL := 1;

	FOR iInitialFL := 1 TO iAddMapArrayLreal DO
			ARBufferlrLrealAddress_Pro[iInitialFL] := ARlrLrealAddress_Pro[iInitialFL];
			ARBufferlrLrealAddress_Hmi[iInitialFL] := ARlrLrealAddress_Pro[iInitialFL];
			ARlrLrealAddress_Hmi[iInitialFL] := ARlrLrealAddress_Pro[iInitialFL];
	END_FOR

END_IF

(*Program*)

			(**********PRO Side Value Change**********)

iProgramFL:= 1;

	FOR iProgramFL := 1 TO iAddMapArrayLreal DO

		ARUpdate_bLrealAddress_Pro[iProgramFL] := FALSE;
		
			IF ARBufferlrLrealAddress_Pro[iProgramFL] <> ARlrLrealAddress_Pro[iProgramFL] THEN
				ARUpdate_bLrealAddress_Pro[iProgramFL] := TRUE;
			END_IF

			IF ARUpdate_bLrealAddress_Pro[iProgramFL] THEN
				ARBufferlrLrealAddress_Pro[iProgramFL] := ARlrLrealAddress_Pro[iProgramFL];
				ARBufferlrLrealAddress_Hmi[iProgramFL] := ARlrLrealAddress_Pro[iProgramFL];
				ARlrLrealAddress_Hmi[iProgramFL] := ARlrLrealAddress_Pro[iProgramFL];
			END_IF
		


					(**********HMI Side Value Change**********)

		ARUpdate_bLrealAddress_Hmi[iProgramFL] := FALSE;

			IF ARBufferlrLrealAddress_Hmi[iProgramFL] <> ARlrLrealAddress_Hmi[iProgramFL] THEN
				ARUpdate_bLrealAddress_Hmi[iProgramFL] := TRUE;
			END_IF
		
			IF ARUpdate_bLrealAddress_Hmi[iProgramFL] THEN
				ARBufferlrLrealAddress_Pro[iProgramFL] := ARlrLrealAddress_Hmi[iProgramFL];
				ARBufferlrLrealAddress_Hmi[iProgramFL] := ARlrLrealAddress_Hmi[iProgramFL];
				ARlrLrealAddress_Pro[iProgramFL] := ARlrLrealAddress_Hmi[iProgramFL];
			END_IF

	END_FOR
(*
(*Lreal 001*)
IF NOT ARUpdate_bLrealAddress_Hmi THEN ARlrLrealAddress_Pro := Pro_lrLreal_001; ELSE Pro_lrLreal_001 := ARlrLrealAddress_Pro; END_IF
IF NOT ARUpdate_bLrealAddress_Pro THEN ARlrLrealAddress_Hmi := Hmi_lrLreal_001; ELSE Hmi_lrLreal_001 := ARlrLrealAddress_Hmi; END_IF
*)

END_FUNCTION_BLOCK

// ---- FBs/B_JKS_NewFB/FBP-HMIAddMapping/fbHMIAddMappingArrayReal.TcPOU
FUNCTION_BLOCK fbHMIAddMappingArrayReal


VAR_INPUT
	bEN : BOOL;
END_VAR
VAR_IN_OUT PERSISTENT
	ARrRealAddress_Pro 					: ARRAY [0..iAddMapArrayReal] OF REAL;
	ARrRealAddress_Hmi 				: ARRAY [0..iAddMapArrayReal] OF REAL;
END_VAR


VAR_OUTPUT
END_VAR


VAR
	ARBufferrRealAddress_Pro 				:  ARRAY [1..iAddMapArrayReal] OF REAL;
	ARBufferrRealAddress_Hmi 				:  ARRAY [1..iAddMapArrayReal] OF REAL;

	ARUpdate_bRealAddress_Pro 				:  ARRAY [1..iAddMapArrayReal] OF BOOL;
	ARUpdate_bRealAddress_Hmi 				:  ARRAY [1..iAddMapArrayReal] OF BOOL;

	iInitialFL: INT;
	iProgramFL: INT;
	bENRE : R_TRIG;


END_VAR

(*Initialized*)
bENRE(CLK:=bEN , Q=> );
IF bENRE.Q THEN
			(*Real*)
iInitialFL := 1;

	FOR iInitialFL := 1 TO iAddMapArrayReal DO
			ARBufferrRealAddress_Pro[iInitialFL] := ARrRealAddress_Pro[iInitialFL];
			ARBufferrRealAddress_Hmi[iInitialFL] := ARrRealAddress_Pro[iInitialFL];
			ARrRealAddress_Hmi[iInitialFL] := ARrRealAddress_Pro[iInitialFL];
	END_FOR

END_IF

(*Program*)

			(**********PRO Side Value Change**********)

iProgramFL:= 1;

	FOR iProgramFL := 1 TO iAddMapArrayReal DO

		ARUpdate_bRealAddress_Pro[iProgramFL] := FALSE;
		
			IF ARBufferrRealAddress_Pro[iProgramFL] <> ARrRealAddress_Pro[iProgramFL] THEN
				ARUpdate_bRealAddress_Pro[iProgramFL] := TRUE;
			END_IF

			IF ARUpdate_bRealAddress_Pro[iProgramFL] THEN
				ARBufferrRealAddress_Pro[iProgramFL] := ARrRealAddress_Pro[iProgramFL];
				ARBufferrRealAddress_Hmi[iProgramFL] := ARrRealAddress_Pro[iProgramFL];
				ARrRealAddress_Hmi[iProgramFL] := ARrRealAddress_Pro[iProgramFL];
			END_IF
		


					(**********HMI Side Value Change**********)
		
		ARUpdate_bRealAddress_Hmi[iProgramFL] := FALSE;

			IF ARBufferrRealAddress_Hmi[iProgramFL] <> ARrRealAddress_Hmi[iProgramFL] THEN
				ARUpdate_bRealAddress_Hmi[iProgramFL] := TRUE;
			END_IF
		
			IF ARUpdate_bRealAddress_Hmi[iProgramFL] THEN
				ARBufferrRealAddress_Pro[iProgramFL] := ARrRealAddress_Hmi[iProgramFL];
				ARBufferrRealAddress_Hmi[iProgramFL] := ARrRealAddress_Hmi[iProgramFL];
				ARrRealAddress_Pro[iProgramFL] := ARrRealAddress_Hmi[iProgramFL];
			END_IF

	END_FOR
(*
(*Real 001*)
IF NOT ARUpdate_bRealAddress_Hmi THEN ARrRealAddress_Pro := Pro_rReal_001; ELSE Pro_rReal_001 := ARrRealAddress_Pro; END_IF
IF NOT ARUpdate_bRealAddress_Pro THEN ARrRealAddress_Hmi := Hmi_rReal_001; ELSE Hmi_rReal_001 := ARrRealAddress_Hmi; END_IF
*)

END_FUNCTION_BLOCK

// ---- FBs/B_JKS_NewFB/FBP-HMIAddMapping/fbHMIAddMappingArrayString.TcPOU
FUNCTION_BLOCK fbHMIAddMappingArrayString


VAR_INPUT
	bEN : BOOL;
END_VAR

VAR_IN_OUT PERSISTENT
	ARsStringAddress_Pro 					: ARRAY [0..iAddMapArrayString] OF STRING;
	ARsStringAddress_Hmi 				: ARRAY [0..iAddMapArrayString] OF STRING;
END_VAR


VAR_OUTPUT
END_VAR


VAR
	ARBuffersStringAddress_Pro 				:  ARRAY [1..iAddMapArrayString] OF STRING;
	ARBuffersStringAddress_Hmi 				:  ARRAY [1..iAddMapArrayString] OF STRING;

	ARUpdate_bStringAddress_Pro 				:  ARRAY [1..iAddMapArrayString] OF BOOL;
	ARUpdate_bStringAddress_Hmi 				:  ARRAY [1..iAddMapArrayString] OF BOOL;

	iInitialFL: INT;
	iProgramFL: INT;
	bENRE : R_TRIG;


END_VAR

(*Initialized*)
bENRE(CLK:=bEN , Q=> );
IF bENRE.Q THEN
			(*String*)
iInitialFL := 1;

	FOR iInitialFL := 1 TO iAddMapArrayString DO
			ARBuffersStringAddress_Pro[iInitialFL] := ARsStringAddress_Pro[iInitialFL];
			ARBuffersStringAddress_Hmi[iInitialFL] := ARsStringAddress_Pro[iInitialFL];
			ARsStringAddress_Hmi[iInitialFL] := ARsStringAddress_Pro[iInitialFL];
	END_FOR

END_IF

(*Program*)

			(**********PRO Side Value Change**********)

iProgramFL:= 1;

	FOR iProgramFL := 1 TO iAddMapArrayString DO

		ARUpdate_bStringAddress_Pro[iProgramFL] := FALSE;

			IF ARBuffersStringAddress_Pro[iProgramFL] <> ARsStringAddress_Pro[iProgramFL] THEN
				ARUpdate_bStringAddress_Pro[iProgramFL] := TRUE;
			END_IF

			IF ARUpdate_bStringAddress_Pro[iProgramFL] THEN
				ARBuffersStringAddress_Pro[iProgramFL] := ARsStringAddress_Pro[iProgramFL];
				ARBuffersStringAddress_Hmi[iProgramFL] := ARsStringAddress_Pro[iProgramFL];
				ARsStringAddress_Hmi[iProgramFL] := ARsStringAddress_Pro[iProgramFL];
			END_IF



					(**********HMI Side Value Change**********)

		ARUpdate_bStringAddress_Hmi[iProgramFL] := FALSE;

			IF ARBuffersStringAddress_Hmi[iProgramFL] <> ARsStringAddress_Hmi[iProgramFL] THEN
				ARUpdate_bStringAddress_Hmi[iProgramFL] := TRUE;
			END_IF

			IF ARUpdate_bStringAddress_Hmi[iProgramFL] THEN
				ARBuffersStringAddress_Pro[iProgramFL] := ARsStringAddress_Hmi[iProgramFL];
				ARBuffersStringAddress_Hmi[iProgramFL] := ARsStringAddress_Hmi[iProgramFL];
				ARsStringAddress_Pro[iProgramFL] := ARsStringAddress_Hmi[iProgramFL];
			END_IF

	END_FOR
(*
(*String 001*)
IF NOT ARUpdate_bStringAddress_Hmi THEN ARsStringAddress_Pro := Pro_sString_001; ELSE Pro_sString_001 := ARsStringAddress_Pro; END_IF
IF NOT ARUpdate_bStringAddress_Pro THEN ARsStringAddress_Hmi := Hmi_sString_001; ELSE Hmi_sString_001 := ARsStringAddress_Hmi; END_IF
*)

END_FUNCTION_BLOCK

// ---- FBs/B_JKS_NewFB/FBP-HMIAddMapping/fbHMIAddMappingBool.TcPOU
FUNCTION_BLOCK fbHMIAddMappingBool


VAR_INPUT
	bEN : BOOL;
END_VAR

VAR_IN_OUT PERSISTENT
	ARbBoolAddress_Pro 					: BOOL;
	ARbBoolAddress_Hmi 				: BOOL;
END_VAR


VAR_OUTPUT
END_VAR


VAR
	ARBufferbBoolAddress_Pro 				:  BOOL;
	ARBufferbBoolAddress_Hmi 				:  BOOL;

	ARUpdate_bBoolAddress_Pro 				:  BOOL;
	ARUpdate_bBoolAddress_Hmi 				:  BOOL;

END_VAR
VAR
	bENRE : R_TRIG;

	ProSideFL: INT;
	HmiSideFL: INT;
END_VAR

(*Initialized*)
bENRE(CLK:=bEN , Q=> );
IF bENRE.Q THEN
			(*Bool*)
			ARBufferbBoolAddress_Pro := ARbBoolAddress_Pro;
			ARBufferbBoolAddress_Hmi := ARbBoolAddress_Pro;
			ARbBoolAddress_Hmi := ARbBoolAddress_Pro;
END_IF

(*Program*)


ARUpdate_bBoolAddress_Pro := FALSE;

	IF ARBufferbBoolAddress_Pro <> ARbBoolAddress_Pro THEN
		ARUpdate_bBoolAddress_Pro := TRUE;
	END_IF

	IF ARUpdate_bBoolAddress_Pro THEN
		ARBufferbBoolAddress_Pro := ARbBoolAddress_Pro;
		ARBufferbBoolAddress_Hmi := ARbBoolAddress_Pro;
		ARbBoolAddress_Hmi := ARbBoolAddress_Pro;
	END_IF



			(**********HMI Side Value Change**********)

ARUpdate_bBoolAddress_Hmi := FALSE;

	(**********Bool**********)
	IF ARBufferbBoolAddress_Hmi <> ARbBoolAddress_Hmi THEN
		ARUpdate_bBoolAddress_Hmi := TRUE;
	END_IF

	IF ARUpdate_bBoolAddress_Hmi THEN
		ARBufferbBoolAddress_Pro := ARbBoolAddress_Hmi;
		ARBufferbBoolAddress_Hmi := ARbBoolAddress_Hmi;
		ARbBoolAddress_Pro := ARbBoolAddress_Hmi;
	END_IF

(*
(*Bool 001*)
IF NOT ARUpdate_bBoolAddress_Hmi THEN ARbBoolAddress_Pro := Pro_bBool_001; ELSE Pro_bBool_001 := ARbBoolAddress_Pro; END_IF
IF NOT ARUpdate_bBoolAddress_Pro THEN ARbBoolAddress_Hmi := Hmi_bBool_001; ELSE Hmi_bBool_001 := ARbBoolAddress_Hmi; END_IF
*)

END_FUNCTION_BLOCK

// ---- FBs/B_JKS_NewFB/FBP-HMIAddMapping/fbHMIAddMappingBoolForManual.TcPOU
FUNCTION_BLOCK fbHMIAddMappingBoolForManual


VAR_INPUT
	bEN : BOOL;
END_VAR

VAR_IN_OUT PERSISTENT
	ARwBoolAddress_Pro 					: WORD;
	ARbBoolAddress_Hmi 				: BOOL;
END_VAR

VAR_OUTPUT
END_VAR


VAR
	ARBufferbBoolAddress_Pro 				:  BOOL;
	ARBufferbBoolAddress_Hmi 				:  BOOL;

	ARUpdate_bBoolAddress_Pro 				:  BOOL;
	ARUpdate_bBoolAddress_Hmi 				:  BOOL;

END_VAR
VAR
	bENRE : R_TRIG;

	ProSideFL: INT;
	HmiSideFL: INT;
END_VAR

(*Initialized*)
bENRE(CLK:=bEN , Q=> );
IF bENRE.Q THEN
			(*Bool*)
			ARBufferbBoolAddress_Pro := ARwBoolAddress_Pro.15;
			ARBufferbBoolAddress_Hmi := ARwBoolAddress_Pro.15;
			ARbBoolAddress_Hmi := ARwBoolAddress_Pro.15;
END_IF

(*Program*)


ARUpdate_bBoolAddress_Pro := FALSE;

	IF ARBufferbBoolAddress_Pro <> ARwBoolAddress_Pro.15 THEN
		ARUpdate_bBoolAddress_Pro := TRUE;
	END_IF

	IF ARUpdate_bBoolAddress_Pro THEN
		ARBufferbBoolAddress_Pro := ARwBoolAddress_Pro.15;
		ARBufferbBoolAddress_Hmi := ARwBoolAddress_Pro.15;
		ARbBoolAddress_Hmi := ARwBoolAddress_Pro.15;
	END_IF



			(**********HMI Side Value Change**********)

ARUpdate_bBoolAddress_Hmi := FALSE;

	(**********Bool**********)
	IF ARBufferbBoolAddress_Hmi <> ARbBoolAddress_Hmi THEN
		ARUpdate_bBoolAddress_Hmi := TRUE;
	END_IF

	IF ARUpdate_bBoolAddress_Hmi THEN
		ARBufferbBoolAddress_Pro := ARbBoolAddress_Hmi;
		ARBufferbBoolAddress_Hmi := ARbBoolAddress_Hmi;
		ARwBoolAddress_Pro.15 := ARbBoolAddress_Hmi;
	END_IF

(*
(*Bool 001*)
IF NOT ARUpdate_bBoolAddress_Hmi THEN ARwBoolAddress_Pro.15 := Pro_bBool_001; ELSE Pro_bBool_001 := ARwBoolAddress_Pro.15; END_IF
IF NOT ARUpdate_bBoolAddress_Pro THEN ARbBoolAddress_Hmi := Hmi_bBool_001; ELSE Hmi_bBool_001 := ARbBoolAddress_Hmi; END_IF
*)

END_FUNCTION_BLOCK

// ---- FBs/B_JKS_NewFB/FBP-HMIAddMapping/fbHMIAddMappingDWordToBoolForManual.TcPOU
FUNCTION_BLOCK fbHMIAddMappingDWordToBoolForManual


VAR_INPUT
	bEN : BOOL;
END_VAR

VAR_IN_OUT PERSISTENT
	ARdwBoolAddress_Pro 					: DWORD;
	ARbBoolAddress_Hmi 				: BOOL;
END_VAR

VAR_OUTPUT
END_VAR


VAR
	ARBufferbBoolAddress_Pro 				:  BOOL;
	ARBufferbBoolAddress_Hmi 				:  BOOL;

	ARUpdate_bBoolAddress_Pro 				:  BOOL;
	ARUpdate_bBoolAddress_Hmi 				:  BOOL;

END_VAR
VAR
	bENRE : R_TRIG;

	ProSideFL: INT;
	HmiSideFL: INT;
END_VAR

(*Initialized*)
bENRE(CLK:=bEN , Q=> );
IF bENRE.Q THEN
			(*Bool*)
			ARBufferbBoolAddress_Pro := ARdwBoolAddress_Pro.31;
			ARBufferbBoolAddress_Hmi := ARdwBoolAddress_Pro.31;
			ARbBoolAddress_Hmi := ARdwBoolAddress_Pro.31;
END_IF

(*Program*)


ARUpdate_bBoolAddress_Pro := FALSE;

	IF ARBufferbBoolAddress_Pro <> ARdwBoolAddress_Pro.31 THEN
		ARUpdate_bBoolAddress_Pro := TRUE;
	END_IF

	IF ARUpdate_bBoolAddress_Pro THEN
		ARBufferbBoolAddress_Pro := ARdwBoolAddress_Pro.31;
		ARBufferbBoolAddress_Hmi := ARdwBoolAddress_Pro.31;
		ARbBoolAddress_Hmi := ARdwBoolAddress_Pro.31;
	END_IF



			(**********HMI Side Value Change**********)

ARUpdate_bBoolAddress_Hmi := FALSE;

	(**********Bool**********)
	IF ARBufferbBoolAddress_Hmi <> ARbBoolAddress_Hmi THEN
		ARUpdate_bBoolAddress_Hmi := TRUE;
	END_IF

	IF ARUpdate_bBoolAddress_Hmi THEN
		ARBufferbBoolAddress_Pro := ARbBoolAddress_Hmi;
		ARBufferbBoolAddress_Hmi := ARbBoolAddress_Hmi;
		ARdwBoolAddress_Pro.31 := ARbBoolAddress_Hmi;
	END_IF

(*
(*Bool 001*)
IF NOT ARUpdate_bBoolAddress_Hmi THEN ARdwBoolAddress_Pro.31 := Pro_bBool_001; ELSE Pro_bBool_001 := ARdwBoolAddress_Pro.31; END_IF
IF NOT ARUpdate_bBoolAddress_Pro THEN ARbBoolAddress_Hmi := Hmi_bBool_001; ELSE Hmi_bBool_001 := ARbBoolAddress_Hmi; END_IF
*)

END_FUNCTION_BLOCK

// ---- FBs/B_JKS_NewFB/FBP-HMIAddMapping/fbHMIAddMappingInt.TcPOU
FUNCTION_BLOCK fbHMIAddMappingInt


VAR_INPUT
	bEN : BOOL;
END_VAR

VAR_IN_OUT PERSISTENT
	ARiIntAddress_Pro 					: INT;
	ARiIntAddress_Hmi 				: INT;
END_VAR


VAR_OUTPUT
END_VAR


VAR
	ARBufferiIntAddress_Pro 				:  INT;
	ARBufferiIntAddress_Hmi 				:  INT;

	ARUpdate_bIntAddress_Pro 				:  BOOL;
	ARUpdate_bIntAddress_Hmi 				:  BOOL;

END_VAR
VAR
	bENRE : R_TRIG;

	ProSideFL: INT;
	HmiSideFL: INT;
END_VAR

(*Initialized*)
bENRE(CLK:=bEN , Q=> );
IF bENRE.Q THEN
			(*Int*)
			ARBufferiIntAddress_Pro := ARiIntAddress_Pro;
			ARBufferiIntAddress_Hmi := ARiIntAddress_Pro;
			ARiIntAddress_Hmi := ARiIntAddress_Pro;
END_IF

(*Program*)


ARUpdate_bIntAddress_Pro := FALSE;

	IF ARBufferiIntAddress_Pro <> ARiIntAddress_Pro THEN
		ARUpdate_bIntAddress_Pro := TRUE;
	END_IF

	IF ARUpdate_bIntAddress_Pro THEN
		ARBufferiIntAddress_Pro := ARiIntAddress_Pro;
		ARBufferiIntAddress_Hmi := ARiIntAddress_Pro;
		ARiIntAddress_Hmi := ARiIntAddress_Pro;
	END_IF



			(**********HMI Side Value Change**********)

ARUpdate_bIntAddress_Hmi := FALSE;

	(**********Int**********)
	IF ARBufferiIntAddress_Hmi <> ARiIntAddress_Hmi THEN
		ARUpdate_bIntAddress_Hmi := TRUE;
	END_IF

	IF ARUpdate_bIntAddress_Hmi THEN
		ARBufferiIntAddress_Pro := ARiIntAddress_Hmi;
		ARBufferiIntAddress_Hmi := ARiIntAddress_Hmi;
		ARiIntAddress_Pro := ARiIntAddress_Hmi;
	END_IF

END_FUNCTION_BLOCK

// ---- FBs/B_JKS_NewFB/FBP-HMIAddMapping/fbHMIAddMappingReal.TcPOU
FUNCTION_BLOCK fbHMIAddMappingReal


VAR_INPUT
	bEN : BOOL;
END_VAR

VAR_IN_OUT PERSISTENT
	ARrRealAddress_Pro 					: REAL;
	ARrRealAddress_Hmi 				: REAL;
END_VAR


VAR_OUTPUT
END_VAR


VAR
	ARBufferrRealAddress_Pro 				:  REAL;
	ARBufferrRealAddress_Hmi 				:  REAL;

	ARUpdate_bRealAddress_Pro 				:  BOOL;
	ARUpdate_bRealAddress_Hmi 				:  BOOL;

END_VAR
VAR
	bENRE : R_TRIG;

	ProSideFL: REAL;
	HmiSideFL: REAL;
END_VAR

(*Initialized*)
bENRE(CLK:=bEN , Q=> );
IF bENRE.Q THEN
			(*Int*)
			ARBufferrRealAddress_Pro := ARrRealAddress_Pro;
			ARBufferrRealAddress_Hmi := ARrRealAddress_Pro;
			ARrRealAddress_Hmi := ARrRealAddress_Pro;
END_IF

(*Program*)


ARUpdate_bRealAddress_Pro := FALSE;

	IF ARBufferrRealAddress_Pro <> ARrRealAddress_Pro THEN
		ARUpdate_bRealAddress_Pro := TRUE;
	END_IF

	IF ARUpdate_bRealAddress_Pro THEN
		ARBufferrRealAddress_Pro := ARrRealAddress_Pro;
		ARBufferrRealAddress_Hmi := ARrRealAddress_Pro;
		ARrRealAddress_Hmi := ARrRealAddress_Pro;
	END_IF



			(**********HMI Side Value Change**********)

ARUpdate_bRealAddress_Hmi := FALSE;

	(**********Int**********)
	IF ARBufferrRealAddress_Hmi <> ARrRealAddress_Hmi THEN
		ARUpdate_bRealAddress_Hmi := TRUE;
	END_IF

	IF ARUpdate_bRealAddress_Hmi THEN
		ARBufferrRealAddress_Pro := ARrRealAddress_Hmi;
		ARBufferrRealAddress_Hmi := ARrRealAddress_Hmi;
		ARrRealAddress_Pro := ARrRealAddress_Hmi;
	END_IF

END_FUNCTION_BLOCK

// ---- FBs/B_JKS_NewFB/FBP-HMIAddMapping/fbHMIAddMappingReal_Int.TcPOU
FUNCTION_BLOCK fbHMIAddMappingReal_Int


VAR_INPUT
	bEN : BOOL;
END_VAR

VAR_IN_OUT PERSISTENT
	ARrRealAddress_Pro 					: REAL;
	ARiIntAddress_Hmi 				: INT;
END_VAR


VAR_OUTPUT
END_VAR


VAR
	ARBufferrRealAddress_Pro 				:  REAL;
	ARBufferiIntAddress_Hmi 					:  INT;

	ARUpdate_bRealAddress_Pro 				:  BOOL;
	ARUpdate_bIntAddress_Hmi 				:  BOOL;

END_VAR
VAR
	bENRE : R_TRIG;

	ProSideFL: REAL;
	HmiSideFL: REAL;
END_VAR

(*Initialized*)
bENRE(CLK:=bEN , Q=> );
IF bENRE.Q THEN
			(*Int*)
			ARBufferrRealAddress_Pro := ARrRealAddress_Pro;
			ARBufferiIntAddress_Hmi := REAL_TO_INT(ARrRealAddress_Pro);
			ARiIntAddress_Hmi := REAL_TO_INT(ARrRealAddress_Pro);
END_IF

(*Program*)


ARUpdate_bRealAddress_Pro := FALSE;

	IF ARBufferrRealAddress_Pro <> ARrRealAddress_Pro THEN
		ARUpdate_bRealAddress_Pro := TRUE;
	END_IF

	IF ARUpdate_bRealAddress_Pro THEN
		ARBufferrRealAddress_Pro := ARrRealAddress_Pro;
		ARBufferiIntAddress_Hmi := REAL_TO_INT(ARrRealAddress_Pro);
		ARiIntAddress_Hmi := REAL_TO_INT(ARrRealAddress_Pro);
	END_IF



			(**********HMI Side Value Change**********)

ARUpdate_bIntAddress_Hmi := FALSE;

	(**********Int**********)
	IF ARBufferiIntAddress_Hmi <> ARiIntAddress_Hmi THEN
		ARUpdate_bIntAddress_Hmi := TRUE;
	END_IF

	IF ARUpdate_bIntAddress_Hmi THEN
		ARBufferrRealAddress_Pro := INT_TO_REAL(ARiIntAddress_Hmi);
		ARBufferiIntAddress_Hmi := ARiIntAddress_Hmi;
		ARrRealAddress_Pro := INT_TO_REAL(ARiIntAddress_Hmi);
	END_IF

END_FUNCTION_BLOCK

// ---- FBs/B_JKS_NewFB/FBP-HMIAddMapping/fbHMIAddMappingString.TcPOU
FUNCTION_BLOCK fbHMIAddMappingString


VAR_INPUT
	bEN : BOOL;
END_VAR

VAR_IN_OUT PERSISTENT
	ARsStringAddress_Pro 					: STRING;
	ARsStringAddress_Hmi 				: STRING;
END_VAR


VAR_OUTPUT
END_VAR


VAR
	ARBuffersStringAddress_Pro 				:  STRING;
	ARBuffersStringAddress_Hmi 				:  STRING;

	ARUpdate_bStringAddress_Pro 				:  BOOL;
	ARUpdate_bStringAddress_Hmi 				:  BOOL;

END_VAR
VAR
	bENRE : R_TRIG;

	ProSideFL: STRING;
	HmiSideFL: STRING;
END_VAR

(*Initialized*)
bENRE(CLK:=bEN , Q=> );
IF bENRE.Q THEN
			(*Int*)
			ARBuffersStringAddress_Pro := ARsStringAddress_Pro;
			ARBuffersStringAddress_Hmi := ARsStringAddress_Pro;
			ARsStringAddress_Hmi := ARsStringAddress_Pro;
END_IF

(*Program*)


ARUpdate_bStringAddress_Pro := FALSE;

	IF ARBuffersStringAddress_Pro <> ARsStringAddress_Pro THEN
		ARUpdate_bStringAddress_Pro := TRUE;
	END_IF

	IF ARUpdate_bStringAddress_Pro THEN
		ARBuffersStringAddress_Pro := ARsStringAddress_Pro;
		ARBuffersStringAddress_Hmi := ARsStringAddress_Pro;
		ARsStringAddress_Hmi := ARsStringAddress_Pro;
	END_IF



			(**********HMI Side Value Change**********)

ARUpdate_bStringAddress_Hmi := FALSE;

	(**********Int**********)
	IF ARBuffersStringAddress_Hmi <> ARsStringAddress_Hmi THEN
		ARUpdate_bStringAddress_Hmi := TRUE;
	END_IF

	IF ARUpdate_bStringAddress_Hmi THEN
		ARBuffersStringAddress_Pro := ARsStringAddress_Hmi;
		ARBuffersStringAddress_Hmi := ARsStringAddress_Hmi;
		ARsStringAddress_Pro := ARsStringAddress_Hmi;
	END_IF

END_FUNCTION_BLOCK

// ---- FBs/B_JKS_NewFB/FBP-HMI/fbScrMapping.TcPOU
FUNCTION_BLOCK fbScrMapping

VAR_INPUT
	iCurrentScrNo : INT;
	bLoadInd : BOOL;
END_VAR

VAR_OUTPUT
END_VAR


VAR

	ScrMapCallSelfCheckRE : R_TRIG;
	iPreviousScrNo : INT;
	ScrMapCallSelfCheckHR : BOOL;
	bInvalidScrMapCallStationSequenceNo : BOOL;
	feScrMapbInvalidCallStationSequenceNo : F_TRIG;
	ScrMapCallStep : INT;
	bScrMapCallCompleted: BOOL;
	InternalTest: BOOL;
	iPreviousScrMapStnSeqRecipeNo: INT;
	ScrMapCallStepSUB: INT;
	iPreviousScrMapStnSubRecipeNo: INT;
	ScrMapCallSelfCheckHRSEQ: BOOL;
	ScrMapCallSelfCheckHRSUB: BOOL;
	iSSERFL: INT;
END_VAR


VAR_IN_OUT PERSISTENT
	ScrMapStnSeqRecipe : DS_fbStationSequenceRecipeStore;
	ScrMapStnSubRecipe : DS_fbStationSubRecipeStore;
	ARStationStnSeqRecipe : ARRAY [0..iStnQty] OF DS_fbStationSequenceRecipeStore;
	ARStationStnSubRecipe : ARRAY [0..iStnQty] OF DS_fbStationSubRecipeStore;



END_VAR

(* Screen Mapping Program*)


ScrMapCallSelfCheckRE(CLK:=iCurrentScrNo <> iPreviousScrNo , Q=> );





IF (*ScrMapCallSelfCheckRE.Q*) iCurrentScrNo <> iPreviousScrNo AND NOT ScrMapCallSelfCheckHR  THEN
ScrMapCallSelfCheckHRSEQ := TRUE;
ScrMapCallSelfCheckHRSUB := TRUE;

END_IF

IF iCurrentScrNo <= 0 OR iCurrentScrNo > iStnQty THEN
bInvalidScrMapCallStationSequenceNo := TRUE;
ELSE
bInvalidScrMapCallStationSequenceNo := FALSE;
END_IF

feScrMapbInvalidCallStationSequenceNo(CLK:=bInvalidScrMapCallStationSequenceNo , Q=> );

(* Mapping for Station SEQUENCE Recipe *)
IF( ScrMapCallSelfCheckRE.Q AND NOT bInvalidScrMapCallStationSequenceNo) OR feScrMapbInvalidCallStationSequenceNo.Q THEN
ScrMapCallStep:= 1;
END_IF


CASE ScrMapCallStep OF

1:
ScrMapStnSeqRecipe := ARStationStnSeqRecipe[iCurrentScrNo];
IF NOT ScrMapCallSelfCheckHRSUB THEN
iPreviousScrNo := iCurrentScrNo;
END_IF
iPreviousScrMapStnSeqRecipeNo := ScrMapStnSeqRecipe.iStationSequenceRecipeNo;
ScrMapCallSelfCheckHRSEQ := FALSE;
ScrMapCallStep := 2;

2:
ARStationStnSeqRecipe[iCurrentScrNo] := ScrMapStnSeqRecipe;

IF iPreviousScrMapStnSeqRecipeNo <> ScrMapStnSeqRecipe.iStationSequenceRecipeNo THEN
ScrMapCallSelfCheckHRSEQ := TRUE;
ScrMapCallStep:= 1;
END_IF

END_CASE


(* Mapping for Station SUB Recipe *)
IF( ScrMapCallSelfCheckRE.Q AND NOT bInvalidScrMapCallStationSequenceNo) OR feScrMapbInvalidCallStationSequenceNo.Q THEN
ScrMapCallStepSUB:= 1;
END_IF


CASE ScrMapCallStepSUB OF

1:
ScrMapStnSubRecipe := ARStationStnSubRecipe[iCurrentScrNo];

iPreviousScrNo := iCurrentScrNo;
iPreviousScrMapStnSubRecipeNo := ScrMapStnSubRecipe.iSubRecipeNo;
ScrMapCallSelfCheckHRSUB := FALSE;
ScrMapCallStepSUB := 2;

2:
ARStationStnSubRecipe[iCurrentScrNo] := ScrMapStnSubRecipe;

IF iPreviousScrMapStnSubRecipeNo <> ScrMapStnSubRecipe.iSubRecipeNo THEN
ScrMapCallSelfCheckHRSUB := TRUE;
ScrMapCallStepSUB:= 1;
END_IF

END_CASE

(*Max and Min Limit*) (*SSER*)
iSSERFL := 1;
FOR iSSERFL := 1 TO iProductRecipeStepArrayQty DO
	IF iSSERFL >= 1 AND iSSERFL <= iProductRecipeStepArrayQty THEN

		IF  ScrMapStnSeqRecipe.DsStationSequenceRecipeMemory.AR10iRepeatFromStepNo[iSSERFL] > iProductRecipeStepArrayQty
		THEN ScrMapStnSeqRecipe.DsStationSequenceRecipeMemory.AR10iRepeatFromStepNo[iSSERFL] := iProductRecipeStepArrayQty;
		ELSIF ScrMapStnSeqRecipe.DsStationSequenceRecipeMemory.AR10iRepeatFromStepNo[iSSERFL] < 1
		THEN ScrMapStnSeqRecipe.DsStationSequenceRecipeMemory.AR10iRepeatFromStepNo[iSSERFL] := 1; END_IF

		IF  ScrMapStnSeqRecipe.DsStationSequenceRecipeMemory.AR10iCycle[iSSERFL] > 99
		THEN ScrMapStnSeqRecipe.DsStationSequenceRecipeMemory.AR10iCycle[iSSERFL] := 99;
		ELSIF ScrMapStnSeqRecipe.DsStationSequenceRecipeMemory.AR10iCycle[iSSERFL] < 1
		THEN ScrMapStnSeqRecipe.DsStationSequenceRecipeMemory.AR10iCycle[iSSERFL] := 1; END_IF

		IF  ScrMapStnSeqRecipe.DsStationSequenceRecipeMemory.AR10iStationSubProNo[iSSERFL] > IStationSubRecipeArrayQty
		THEN ScrMapStnSeqRecipe.DsStationSequenceRecipeMemory.AR10iStationSubProNo[iSSERFL] := IStationSubRecipeArrayQty;
		ELSIF ScrMapStnSeqRecipe.DsStationSequenceRecipeMemory.AR10iStationSubProNo[iSSERFL] < 0
		THEN ScrMapStnSeqRecipe.DsStationSequenceRecipeMemory.AR10iStationSubProNo[iSSERFL] := 0; END_IF

	END_IF
END_FOR



(*Max and Min Limit*) (*SSUR*)
IF  ScrMapStnSubRecipe.DsSubRecipeMemory.iStCon1TargetVacuumLevel > 101 THEN ScrMapStnSubRecipe.DsSubRecipeMemory.iStCon1TargetVacuumLevel := 101; ELSIF ScrMapStnSubRecipe.DsSubRecipeMemory.iStCon1TargetVacuumLevel < -101 THEN ScrMapStnSubRecipe.DsSubRecipeMemory.iStCon1TargetVacuumLevel := -101; END_IF
IF  ScrMapStnSubRecipe.DsSubRecipeMemory.iStCon2TargetPressureLevel > 101 THEN ScrMapStnSubRecipe.DsSubRecipeMemory.iStCon2TargetPressureLevel := 101; ELSIF ScrMapStnSubRecipe.DsSubRecipeMemory.iStCon2TargetPressureLevel < -101 THEN ScrMapStnSubRecipe.DsSubRecipeMemory.iStCon2TargetPressureLevel := -101; END_IF
IF  ScrMapStnSubRecipe.DsSubRecipeMemory.iStCon3TargetProTankTempLevel > 200 THEN ScrMapStnSubRecipe.DsSubRecipeMemory.iStCon3TargetProTankTempLevel := 200; ELSIF ScrMapStnSubRecipe.DsSubRecipeMemory.iStCon3TargetProTankTempLevel < 20 THEN ScrMapStnSubRecipe.DsSubRecipeMemory.iStCon3TargetProTankTempLevel := 20; END_IF
IF  ScrMapStnSubRecipe.DsSubRecipeMemory.iStCon4TargetSubTankTempLevel > 200 THEN ScrMapStnSubRecipe.DsSubRecipeMemory.iStCon4TargetSubTankTempLevel := 200; ELSIF ScrMapStnSubRecipe.DsSubRecipeMemory.iStCon4TargetSubTankTempLevel < 20 THEN ScrMapStnSubRecipe.DsSubRecipeMemory.iStCon4TargetSubTankTempLevel := 20; END_IF

IF  ScrMapStnSubRecipe.DsSubRecipeMemory.iComCon1TargetVacuumLevel > 101 THEN ScrMapStnSubRecipe.DsSubRecipeMemory.iComCon1TargetVacuumLevel := 101; ELSIF ScrMapStnSubRecipe.DsSubRecipeMemory.iComCon1TargetVacuumLevel < -101 THEN ScrMapStnSubRecipe.DsSubRecipeMemory.iComCon1TargetVacuumLevel := -101; END_IF
IF  ScrMapStnSubRecipe.DsSubRecipeMemory.iComCon2TargetPressureLevel > 101 THEN ScrMapStnSubRecipe.DsSubRecipeMemory.iComCon2TargetPressureLevel := 101; ELSIF ScrMapStnSubRecipe.DsSubRecipeMemory.iComCon2TargetPressureLevel < -101 THEN ScrMapStnSubRecipe.DsSubRecipeMemory.iComCon2TargetPressureLevel := -101; END_IF
IF  ScrMapStnSubRecipe.DsSubRecipeMemory.iComCon3TargetProTankTempLevel > 200 THEN ScrMapStnSubRecipe.DsSubRecipeMemory.iComCon3TargetProTankTempLevel := 200; ELSIF ScrMapStnSubRecipe.DsSubRecipeMemory.iComCon3TargetProTankTempLevel < 20 THEN ScrMapStnSubRecipe.DsSubRecipeMemory.iComCon3TargetProTankTempLevel := 20; END_IF
IF  ScrMapStnSubRecipe.DsSubRecipeMemory.iComCon4TargetSubTankTempLevel > 200 THEN ScrMapStnSubRecipe.DsSubRecipeMemory.iComCon4TargetSubTankTempLevel := 200; ELSIF ScrMapStnSubRecipe.DsSubRecipeMemory.iComCon4TargetSubTankTempLevel < 20 THEN ScrMapStnSubRecipe.DsSubRecipeMemory.iComCon4TargetSubTankTempLevel := 20; END_IF

IF  ScrMapStnSubRecipe.DsSubRecipeMemory.iComCon5ProcessTimer > 9999 THEN ScrMapStnSubRecipe.DsSubRecipeMemory.iComCon5ProcessTimer := 9999; ELSIF ScrMapStnSubRecipe.DsSubRecipeMemory.iComCon5ProcessTimer < 0 THEN ScrMapStnSubRecipe.DsSubRecipeMemory.iComCon5ProcessTimer := 0; END_IF

IF  ScrMapStnSubRecipe.DsSubRecipeMemory.iOut1ProTankPumpLPM > 999 THEN ScrMapStnSubRecipe.DsSubRecipeMemory.iOut1ProTankPumpLPM := 999; ELSIF ScrMapStnSubRecipe.DsSubRecipeMemory.iOut1ProTankPumpLPM < 0 THEN ScrMapStnSubRecipe.DsSubRecipeMemory.iOut1ProTankPumpLPM := 0; END_IF

IF  ScrMapStnSubRecipe.DsSubRecipeMemory.iOut2ProTankPumpHz > 300 THEN ScrMapStnSubRecipe.DsSubRecipeMemory.iOut2ProTankPumpHz := 300; ELSIF ScrMapStnSubRecipe.DsSubRecipeMemory.iOut2ProTankPumpHz < 0 THEN ScrMapStnSubRecipe.DsSubRecipeMemory.iOut2ProTankPumpHz := 0; END_IF

IF  ScrMapStnSubRecipe.DsSubRecipeMemory.iOut3ProTankBtmUsAPwrPercent > 100 THEN ScrMapStnSubRecipe.DsSubRecipeMemory.iOut3ProTankBtmUsAPwrPercent := 100; ELSIF ScrMapStnSubRecipe.DsSubRecipeMemory.iOut3ProTankBtmUsAPwrPercent < 10 THEN ScrMapStnSubRecipe.DsSubRecipeMemory.iOut3ProTankBtmUsAPwrPercent := 10; END_IF
IF  ScrMapStnSubRecipe.DsSubRecipeMemory.iOut4ProTankBtmUsBPwrPercent > 100 THEN ScrMapStnSubRecipe.DsSubRecipeMemory.iOut4ProTankBtmUsBPwrPercent := 100; ELSIF ScrMapStnSubRecipe.DsSubRecipeMemory.iOut4ProTankBtmUsBPwrPercent < 10 THEN ScrMapStnSubRecipe.DsSubRecipeMemory.iOut4ProTankBtmUsBPwrPercent := 10; END_IF
IF  ScrMapStnSubRecipe.DsSubRecipeMemory.iOut5ProTankBtmUsCPwrPercent > 100 THEN ScrMapStnSubRecipe.DsSubRecipeMemory.iOut5ProTankBtmUsCPwrPercent := 100; ELSIF ScrMapStnSubRecipe.DsSubRecipeMemory.iOut5ProTankBtmUsCPwrPercent < 10 THEN ScrMapStnSubRecipe.DsSubRecipeMemory.iOut5ProTankBtmUsCPwrPercent := 10; END_IF
IF  ScrMapStnSubRecipe.DsSubRecipeMemory.iOut6ProTankSideUsAPwrPercent > 100 THEN ScrMapStnSubRecipe.DsSubRecipeMemory.iOut6ProTankSideUsAPwrPercent := 100; ELSIF ScrMapStnSubRecipe.DsSubRecipeMemory.iOut6ProTankSideUsAPwrPercent < 10 THEN ScrMapStnSubRecipe.DsSubRecipeMemory.iOut6ProTankSideUsAPwrPercent := 10; END_IF
IF  ScrMapStnSubRecipe.DsSubRecipeMemory.iOut7ProTankSideUsBPwrPercent > 100 THEN ScrMapStnSubRecipe.DsSubRecipeMemory.iOut7ProTankSideUsBPwrPercent := 100; ELSIF ScrMapStnSubRecipe.DsSubRecipeMemory.iOut7ProTankSideUsBPwrPercent < 10 THEN ScrMapStnSubRecipe.DsSubRecipeMemory.iOut7ProTankSideUsBPwrPercent := 10; END_IF
(*
IF  ScrMapStnSubRecipe.DsSubRecipeMemory.iOut8ProTankBtmUsAkHz > 500 THEN ScrMapStnSubRecipe.DsSubRecipeMemory.iOut8ProTankBtmUsAkHz := 500; ELSIF ScrMapStnSubRecipe.DsSubRecipeMemory.iOut8ProTankBtmUsAkHz < 25 THEN ScrMapStnSubRecipe.DsSubRecipeMemory.iOut8ProTankBtmUsAkHz := 25; END_IF
IF  ScrMapStnSubRecipe.DsSubRecipeMemory.iOut9ProTankBtmUsBkHz > 500 THEN ScrMapStnSubRecipe.DsSubRecipeMemory.iOut9ProTankBtmUsBkHz := 500; ELSIF ScrMapStnSubRecipe.DsSubRecipeMemory.iOut9ProTankBtmUsBkHz < 25 THEN ScrMapStnSubRecipe.DsSubRecipeMemory.iOut9ProTankBtmUsBkHz := 25; END_IF
IF  ScrMapStnSubRecipe.DsSubRecipeMemory.iOut10ProTankBtmUsCkHz > 500 THEN ScrMapStnSubRecipe.DsSubRecipeMemory.iOut10ProTankBtmUsCkHz := 500; ELSIF ScrMapStnSubRecipe.DsSubRecipeMemory.iOut10ProTankBtmUsCkHz < 25 THEN ScrMapStnSubRecipe.DsSubRecipeMemory.iOut10ProTankBtmUsCkHz := 25; END_IF
IF  ScrMapStnSubRecipe.DsSubRecipeMemory.iOut11ProTankSideUsAkHz > 500 THEN ScrMapStnSubRecipe.DsSubRecipeMemory.iOut11ProTankSideUsAkHz := 500; ELSIF ScrMapStnSubRecipe.DsSubRecipeMemory.iOut11ProTankSideUsAkHz < 25 THEN ScrMapStnSubRecipe.DsSubRecipeMemory.iOut11ProTankSideUsAkHz := 25; END_IF
IF  ScrMapStnSubRecipe.DsSubRecipeMemory.iOut12ProTankSideUsBkHz > 500 THEN ScrMapStnSubRecipe.DsSubRecipeMemory.iOut12ProTankSideUsBkHz := 500; ELSIF ScrMapStnSubRecipe.DsSubRecipeMemory.iOut12ProTankSideUsBkHz < 25 THEN ScrMapStnSubRecipe.DsSubRecipeMemory.iOut12ProTankSideUsBkHz := 25; END_IF
*)
IF  ScrMapStnSubRecipe.DsSubRecipeMemory.iOut13ProTankBlowerHz > 300 THEN ScrMapStnSubRecipe.DsSubRecipeMemory.iOut13ProTankBlowerHz := 300; ELSIF ScrMapStnSubRecipe.DsSubRecipeMemory.iOut13ProTankBlowerHz < 40 THEN ScrMapStnSubRecipe.DsSubRecipeMemory.iOut13ProTankBlowerHz := 40; END_IF

IF  ScrMapStnSubRecipe.DsSubRecipeMemory.rOut14ProTankChangeTemperatureDegC > 200 THEN ScrMapStnSubRecipe.DsSubRecipeMemory.rOut14ProTankChangeTemperatureDegC := 200; ELSIF ScrMapStnSubRecipe.DsSubRecipeMemory.rOut14ProTankChangeTemperatureDegC < 20 THEN ScrMapStnSubRecipe.DsSubRecipeMemory.rOut14ProTankChangeTemperatureDegC := 20; END_IF
IF  ScrMapStnSubRecipe.DsSubRecipeMemory.rOut15SubTankChangeTemperatureDegC > 200 THEN ScrMapStnSubRecipe.DsSubRecipeMemory.rOut15SubTankChangeTemperatureDegC := 200; ELSIF ScrMapStnSubRecipe.DsSubRecipeMemory.rOut15SubTankChangeTemperatureDegC < 20 THEN ScrMapStnSubRecipe.DsSubRecipeMemory.rOut15SubTankChangeTemperatureDegC := 20; END_IF


IF  ScrMapStnSubRecipe.DsSubRecipeMemory.iOut16SubTankPumpLPM > 999 THEN ScrMapStnSubRecipe.DsSubRecipeMemory.iOut16SubTankPumpLPM := 999; ELSIF ScrMapStnSubRecipe.DsSubRecipeMemory.iOut16SubTankPumpLPM < 0 THEN ScrMapStnSubRecipe.DsSubRecipeMemory.iOut16SubTankPumpLPM := 0; END_IF

IF  ScrMapStnSubRecipe.DsSubRecipeMemory.iOut17SubTankPumpHz > 300 THEN ScrMapStnSubRecipe.DsSubRecipeMemory.iOut17SubTankPumpHz := 300; ELSIF ScrMapStnSubRecipe.DsSubRecipeMemory.iOut17SubTankPumpHz < 0 THEN ScrMapStnSubRecipe.DsSubRecipeMemory.iOut17SubTankPumpHz := 0; END_IF

IF  ScrMapStnSubRecipe.DsSubRecipeMemory.iOut18SlowPullVelocity > 50 THEN ScrMapStnSubRecipe.DsSubRecipeMemory.iOut18SlowPullVelocity := 50; ELSIF ScrMapStnSubRecipe.DsSubRecipeMemory.iOut18SlowPullVelocity < 1 THEN ScrMapStnSubRecipe.DsSubRecipeMemory.iOut18SlowPullVelocity := 1; END_IF

END_FUNCTION_BLOCK

// ---- FBs/B_JKS_NewFB/FBP-Instrument/fbClangsonicUltrasonic.TcPOU
FUNCTION_BLOCK fbClangsonicUltrasonic
VAR_INPUT

	bStart: BOOL;

	wModbusStartAddress: WORD;

	ARbyUnitID: ARRAY [1..iUSGeneratorQty] OF BYTE;

END_VAR
VAR_IN_OUT PERSISTENT
	DSClangsonicGenerator : ARRAY [1..iUSGeneratorQty] OF DS_ClangsonicGenerator;

END_VAR
VAR_OUTPUT
	bModbusBusy: BOOL;
	bModbusError: BOOL;

END_VAR
VAR
	ClangsonicModbus:ModbusRtuMaster_KL6x22B;

	bModbusReadStRE: R_TRIG;
	bModbusWriteStRE: R_TRIG;
	bStartRE: R_TRIG;

	bModbusReadSt: BOOL;
	bModbusWriteSt: BOOL;

	iStep: INT;
	iIDCounter: INT;
	iAddCounter: INT;

	iMFL: INT;
	iSFL: INT;

	bInternalTestPB : BOOL;

	bInternalTestPBRE: R_TRIG;
	ErrorId_Read: MODBUS_ERRORS;
	ErrorId_Write: MODBUS_ERRORS;
END_VAR
VAR PERSISTENT

	AR2SwModbusReadData: ARRAY [1..iUSGeneratorQty, 1..iModbusRWQty] OF WORD;
(*	AR2SwModbusWriteData: ARRAY [1..iUSGeneratorQty, 1..iModbusRWQty] OF WORD;*)

	AR2SwModbusReadDataBuffer: ARRAY [1..iUSGeneratorQty, 1..iModbusRWQty] OF WORD;
	AR2SwModbusWriteDataBuffer: ARRAY [1..iUSGeneratorQty, 1..iModbusRWQty] OF WORD;

	AR2SbWriteInProgress: ARRAY [1..iUSGeneratorQty, 1..iModbusRWQty] OF BOOL;


END_VAR

(* Min/Max Ctrl*)
IF iIDCounter > iUSGeneratorQty THEN
iIDCounter := iUSGeneratorQty;
ELSIF iIDCounter < 1 THEN
iIDCounter := 1;
END_IF

IF iAddCounter > iModbusRWQty THEN
iAddCounter := iModbusRWQty;
ELSIF iAddCounter < 1 THEN
iAddCounter := 1;
END_IF

(*Address Mapping*)

iMFL := 1;
	FOR iMFL := 1 TO iUSGeneratorQty DO
		IF iMFL >= 1 AND iMFL <= iUSGeneratorQty THEN
			iSFL :=1;
				FOR iSFL := 1 TO iModbusRWQty DO
					IF iSFL >= 1 AND iSFL <= iModbusRWQty THEN
						IF ( (AR2SwModbusReadData[iMFL,iSFL] <> AR2SwModbusReadDataBuffer[iMFL,iSFL])
						AND NOT AR2SbWriteInProgress[iMFL,iSFL])
						OR (NOT DSClangsonicGenerator[iMFL].bModbusWriteEn[iSFL])
						THEN
							DSClangsonicGenerator[iMFL].wModbusData[iSFL] 	:= AR2SwModbusReadData[iMFL,iSFL];
							(*AR2SwModbusWriteData[iMFL,iSFL] 				:= AR2SwModbusReadData[iMFL,iSFL];*)
							AR2SwModbusReadDataBuffer[iMFL,iSFL] 			:= AR2SwModbusReadData[iMFL,iSFL];
							AR2SwModbusWriteDataBuffer[iMFL,iSFL] 			:= AR2SwModbusReadData[iMFL,iSFL];


						END_IF

						IF NOT DSClangsonicGenerator[iMFL].bModbusWriteEn[iSFL]
						AND DSClangsonicGenerator[iMFL].wModbusData[iSFL] <> AR2SwModbusWriteDataBuffer[iMFL,iSFL]
						THEN
							(*AR2SwModbusReadData[iMFL,iSFL] 			 	:= DSClangsonicGenerator[iMFL].wModbusData[iSFL];*)
							(*AR2SwModbusReadData[iMFL,iSFL] 			 	:= DSClangsonicGenerator[iMFL].wModbusData[iSFL];
							AR2SwModbusReadDataBuffer[iMFL,iSFL] 			:= DSClangsonicGenerator[iMFL].wModbusData[iSFL];
							*)AR2SwModbusWriteDataBuffer[iMFL,iSFL] 			:= DSClangsonicGenerator[iMFL].wModbusData[iSFL];

							AR2SbWriteInProgress[iMFL,iSFL] := TRUE;
						END_IF
					END_IF
				END_FOR
		END_IF
	END_FOR


(*Read / Write*)
bInternalTestPBRE(CLK:=bInternalTestPB , Q=> );
bStartRE(CLK:=bStart , Q=> );
IF bStartRE.Q OR bInternalTestPBRE.Q THEN
iStep := 1;
END_IF
IF NOT bStart AND NOT bInternalTestPB THEN
iStep := 0;
END_IF

bModbusReadStRE(CLK:=bModbusReadSt , Q=> );
bModbusWriteStRE(CLK:=bModbusWriteSt , Q=> );


ClangsonicModbus.ReadRegs(
	UnitID:=ARbyUnitID[iIDCounter] ,
	Quantity:= 1(*INT_TO_WORD(iModbusRWQty)*),
	MBAddr:= wModbusStartAddress+iAddCounter-1,
	cbLength:= SIZEOF(AR2SwModbusReadData[iIDCounter,iAddCounter]),
	pMemoryAddr:= ADR(AR2SwModbusReadData[iIDCounter,iAddCounter]),
	Execute:= bModbusReadStRE.Q,
	Timeout:= t#2s,
	BUSY=> bModbusBusy,
	Error=> bModbusError,
	ErrorId=>ErrorId_Read ,
	cbRead=> );

ClangsonicModbus.WriteSingleRegister(
	UnitID:=ARbyUnitID[iIDCounter] ,
	Quantity:= 1,
	MBAddr:= wModbusStartAddress+iAddCounter-1,
	cbLength:= SIZEOF(DSClangsonicGenerator[iIDCounter].wModbusData[iAddCounter]),
	pMemoryAddr:= ADR((*AR2SwModbusWriteData[iIDCounter,iAddCounter]*)DSClangsonicGenerator[iIDCounter].wModbusData[iAddCounter]),
	Execute:= bModbusWriteStRE.Q,
	Timeout:= t#2s,
	BUSY=> bModbusBusy,
	Error=> bModbusError,
	ErrorId=>ErrorId_Write ,
	cbRead=> );


CASE iStep OF
0:
bModbusReadSt := FALSE;
bModbusWriteSt := FALSE;

1: (*Read Data*)
IF bModbusReadSt AND NOT bModbusBusy
OR AR2SbWriteInProgress[iIDCounter,iAddCounter]
THEN
	IF iAddCounter < iModbusRWQty THEN

		iAddCounter := iAddCounter + 1;

	ELSIF iAddCounter >= iModbusRWQty THEN

			IF iIDCounter < iUSGeneratorQty THEN
				iIDCounter := iIDCounter + 1;
			ELSIF iIDCounter >= iUSGeneratorQty THEN
				iIDCounter := 1;
			END_IF

		iAddCounter := 1;
	END_IF


(*DSClangsonicGenerator[iIDCounter].wModbusData[iAddCounter] := AR2SwModbusReadData[iIDCounter,iAddCounter];*)
iStep := 2;

END_IF

IF NOT AR2SbWriteInProgress[iIDCounter,iAddCounter]  THEN
bModbusReadSt := TRUE;
bModbusWriteSt := FALSE;
END_IF

2: (*Write Data*)
IF (bModbusWriteSt AND NOT bModbusBusy)
OR (AR2SwModbusReadData[iIDCounter,iAddCounter] = DSClangsonicGenerator[iIDCounter].wModbusData[iAddCounter])
OR NOT DSClangsonicGenerator[iIDCounter].bModbusWriteEn[iAddCounter]
 THEN
iStep := 1;
AR2SbWriteInProgress[iIDCounter,iAddCounter] := FALSE;

bModbusReadSt := FALSE;
bModbusWriteSt := FALSE;
END_IF

IF (AR2SwModbusReadData[iIDCounter,iAddCounter] <> DSClangsonicGenerator[iIDCounter].wModbusData[iAddCounter])
AND DSClangsonicGenerator[iIDCounter].bModbusWriteEn[iAddCounter]
THEN
(*DSClangsonicGenerator[iIDCounter].wModbusData[iAddCounter] := AR2SwModbusReadData[iIDCounter,iAddCounter];*)

bModbusReadSt := FALSE;
bModbusWriteSt := TRUE;
END_IF

END_CASE

END_FUNCTION_BLOCK

// ---- FBs/B_JKS_NewFB/FBP-Instrument/fbClangsonicUltrasonic_test.TcPOU
FUNCTION_BLOCK fbClangsonicUltrasonic_test
VAR_INPUT

	bStart: BOOL;

	wModbusStartAddress: WORD;

	ARbyUnitID: ARRAY [1..iUSGeneratorQty] OF BYTE;

END_VAR
VAR_IN_OUT PERSISTENT
	DSClangsonicGenerator : ARRAY [1..iUSGeneratorQty] OF DS_ClangsonicGenerator;

END_VAR
VAR_OUTPUT
	bModbusBusy: BOOL;
	bModbusError: BOOL;

END_VAR
VAR
	ClangsonicModbus:ModbusRtuMaster_KL6x22B;

	bModbusReadStRE: R_TRIG;
	bModbusWriteStRE: R_TRIG;
	bStartRE: R_TRIG;

	bModbusReadSt: BOOL;
	bModbusWriteSt: BOOL;

	iStep: INT;
	iIDCounter: INT;
	iAddCounter: INT;

	iMFL: INT;
	iSFL: INT;

	bInternalTestPB : BOOL;

	bInternalTestPBRE: R_TRIG;
	ErrorId_Read: MODBUS_ERRORS;
	ErrorId_Write: MODBUS_ERRORS;
END_VAR
VAR PERSISTENT

	AR2SwModbusReadData: ARRAY [1..iUSGeneratorQty, 1..iModbusRWQty] OF WORD;
(*	AR2SwModbusWriteData: ARRAY [1..iUSGeneratorQty, 1..iModbusRWQty] OF WORD;*)

	AR2SwModbusReadDataBuffer: ARRAY [1..iUSGeneratorQty, 1..iModbusRWQty] OF WORD;
	AR2SwModbusWriteDataBuffer: ARRAY [1..iUSGeneratorQty, 1..iModbusRWQty] OF WORD;

	AR2SbWriteInProgress: ARRAY [1..iUSGeneratorQty, 1..iModbusRWQty] OF BOOL;


END_VAR

(* Min/Max Ctrl*)
IF iIDCounter > iUSGeneratorQty THEN
iIDCounter := iUSGeneratorQty;
ELSIF iIDCounter < 1 THEN
iIDCounter := 1;
END_IF

IF iAddCounter > iModbusRWQty THEN
iAddCounter := iModbusRWQty;
ELSIF iAddCounter < 1 THEN
iAddCounter := 1;
END_IF

(*Address Mapping*)

iMFL := 1;
	FOR iMFL := 1 TO iUSGeneratorQty DO
		IF iMFL >= 1 AND iMFL <= iUSGeneratorQty THEN
			iSFL :=1;
				FOR iSFL := 1 TO iModbusRWQty DO
					IF iSFL >= 1 AND iSFL <= iModbusRWQty THEN
						IF ( (AR2SwModbusReadData[iMFL,iSFL] <> AR2SwModbusReadDataBuffer[iMFL,iSFL])
						AND NOT AR2SbWriteInProgress[iMFL,iSFL])
						OR (NOT DSClangsonicGenerator[iMFL].bModbusWriteEn[iSFL])
						THEN
							DSClangsonicGenerator[iMFL].wModbusData[iSFL] 	:= AR2SwModbusReadData[iMFL,iSFL];
							(*AR2SwModbusWriteData[iMFL,iSFL] 				:= AR2SwModbusReadData[iMFL,iSFL];*)
							AR2SwModbusReadDataBuffer[iMFL,iSFL] 			:= AR2SwModbusReadData[iMFL,iSFL];
							AR2SwModbusWriteDataBuffer[iMFL,iSFL] 			:= AR2SwModbusReadData[iMFL,iSFL];


						END_IF

						IF NOT DSClangsonicGenerator[iMFL].bModbusWriteEn[iSFL]
						AND DSClangsonicGenerator[iMFL].wModbusData[iSFL] <> AR2SwModbusWriteDataBuffer[iMFL,iSFL]
						THEN
							(*AR2SwModbusReadData[iMFL,iSFL] 			 	:= DSClangsonicGenerator[iMFL].wModbusData[iSFL];*)
							(*AR2SwModbusReadData[iMFL,iSFL] 			 	:= DSClangsonicGenerator[iMFL].wModbusData[iSFL];
							AR2SwModbusReadDataBuffer[iMFL,iSFL] 			:= DSClangsonicGenerator[iMFL].wModbusData[iSFL];
							*)AR2SwModbusWriteDataBuffer[iMFL,iSFL] 			:= DSClangsonicGenerator[iMFL].wModbusData[iSFL];

							AR2SbWriteInProgress[iMFL,iSFL] := TRUE;
						END_IF
					END_IF
				END_FOR
		END_IF
	END_FOR


(*Read / Write*)
bInternalTestPBRE(CLK:=bInternalTestPB , Q=> );
bStartRE(CLK:=bStart , Q=> );
IF bStartRE.Q OR bInternalTestPBRE.Q THEN
iStep := 1;
END_IF
IF NOT bStart AND NOT bInternalTestPB THEN
iStep := 0;
END_IF

bModbusReadStRE(CLK:=bModbusReadSt , Q=> );
bModbusWriteStRE(CLK:=bModbusWriteSt , Q=> );


ClangsonicModbus.ReadRegs(
	UnitID:=ARbyUnitID[iIDCounter] ,
	Quantity:= 1(*INT_TO_WORD(iModbusRWQty)*),
	MBAddr:= wModbusStartAddress+iAddCounter-1,
	cbLength:= SIZEOF(AR2SwModbusReadData[iIDCounter,iAddCounter]),
	pMemoryAddr:= ADR(AR2SwModbusReadData[iIDCounter,iAddCounter]),
	Execute:= bModbusReadStRE.Q,
	Timeout:= t#2s,
	BUSY=> bModbusBusy,
	Error=> bModbusError,
	ErrorId=>ErrorId_Read ,
	cbRead=> );

ClangsonicModbus.WriteSingleRegister(
	UnitID:=ARbyUnitID[iIDCounter] ,
	Quantity:= 1,
	MBAddr:= wModbusStartAddress+iAddCounter-1,
	cbLength:= SIZEOF(DSClangsonicGenerator[iIDCounter].wModbusData[iAddCounter]),
	pMemoryAddr:= ADR((*AR2SwModbusWriteData[iIDCounter,iAddCounter]*)DSClangsonicGenerator[iIDCounter].wModbusData[iAddCounter]),
	Execute:= bModbusWriteStRE.Q,
	Timeout:= t#2s,
	BUSY=> bModbusBusy,
	Error=> bModbusError,
	ErrorId=>ErrorId_Write ,
	cbRead=> );


CASE iStep OF
0:
bModbusReadSt := FALSE;
bModbusWriteSt := FALSE;

1: (*Read Data*)
IF bModbusReadSt AND NOT bModbusBusy
OR AR2SbWriteInProgress[iIDCounter,iAddCounter]
THEN
	IF iAddCounter < iModbusRWQty THEN

		iAddCounter := iAddCounter + 1;

	ELSIF iAddCounter >= iModbusRWQty THEN

			IF iIDCounter < iUSGeneratorQty THEN
				iIDCounter := iIDCounter + 1;
			ELSIF iIDCounter >= iUSGeneratorQty THEN
				iIDCounter := 1;
			END_IF

		iAddCounter := 1;
	END_IF


(*DSClangsonicGenerator[iIDCounter].wModbusData[iAddCounter] := AR2SwModbusReadData[iIDCounter,iAddCounter];*)
iStep := 2;

END_IF

IF NOT AR2SbWriteInProgress[iIDCounter,iAddCounter]  THEN
bModbusReadSt := TRUE;
bModbusWriteSt := FALSE;
END_IF

2: (*Write Data*)
IF (bModbusWriteSt AND NOT bModbusBusy)
OR (AR2SwModbusReadData[iIDCounter,iAddCounter] = DSClangsonicGenerator[iIDCounter].wModbusData[iAddCounter])
OR NOT DSClangsonicGenerator[iIDCounter].bModbusWriteEn[iAddCounter]
 THEN
iStep := 1;
AR2SbWriteInProgress[iIDCounter,iAddCounter] := FALSE;

bModbusReadSt := FALSE;
bModbusWriteSt := FALSE;
END_IF

IF (AR2SwModbusReadData[iIDCounter,iAddCounter] <> DSClangsonicGenerator[iIDCounter].wModbusData[iAddCounter])
AND DSClangsonicGenerator[iIDCounter].bModbusWriteEn[iAddCounter]
THEN
(*DSClangsonicGenerator[iIDCounter].wModbusData[iAddCounter] := AR2SwModbusReadData[iIDCounter,iAddCounter];*)

bModbusReadSt := FALSE;
bModbusWriteSt := TRUE;
END_IF

END_CASE

END_FUNCTION_BLOCK

// ---- FBs/B_JKS_NewFB/FBP-Memory_Sub/fbGnrStationMasterController.TcPOU
FUNCTION_BLOCK fbGnrStationMasterController

VAR_INPUT
	bTrackerEN								: BOOL;
	bTrackerBasedOnPreviousTime			: BOOL;
	iCurrentStationAddress 					: INT;															(* Input - Define current station no so that this fb know which array number to used*)
	iPreCallArmTime							: INT;															(* Input - Pre-Call Arm Time, Program will call arm if the Total process timeEV Equal or Lesser than this value*)
	iTotalProcessTimeSV						:INT;
	iCurrentStnSeqProcessTotalTime 		: INT;															(* Input - Link with fbStnSeqProcess, to collect CurrentProcessTotalTime*)
	iPreviousStnSeqProcessTotalTime 		: INT; 															(* Input - Link with fbStnSeqProcess,  to collect PreviousProcessTotalTime*)
	bStnSeqProcessInProgressFlag			: BOOL;														(* Input - Link with fbStnSeqProcess,  to collect the status of process in progress from StnSeqProcessfb*)
	bStnSeqProcessCompleted 				: BOOL;														(* Input - Link with fbStnSeqProcess,  to collect the status of process completion from StnSeqProcessfb*)
	ARbAlternateStnEn : ARRAY [1..iAlternateSetQty] OF BOOL;
	AR2siAlternateStn : ARRAY [1..iAlternateSetQty, 1..iAlternateStnQty] OF INT;
(*	DSStnSeqProOutput 				:DS_StnSeqProOutput;								(* Output - To Control Output - When process running, instrument should control by the output in this Data structure*)
*)

END_VAR

VAR_IN_OUT PERSISTENT
	bStnSeqProcessSt						: BOOL;														(* Output - Link with fbStnSeqProcess, After Read out from fbGnrProductRecipeMemory, this fb will trigger this Bool to start the StnSeqProcess*)

	ARbProductRecipeCallEn 				: ARRAY [0..iStnQty] OF BOOL;					(* Output - Link with fbGnrProductRecipeMemory, Array based on Current Station No, the fbGnrProductRecipeMemory will start Read info from Memory when this bool turn on*)
	ARiProductRecipeNoCall 				: ARRAY [0..iStnQty] OF INT;						(* Output - Link with fbGnrProductRecipeMemory, Array based on Current Station No, the read out from fbGnrProductRecipeMemory is based on this Product Recipe No*)
	ARiProductRecipeStepCall 				: ARRAY [0..iStnQty] OF INT;						(* Output - Link with fbGnrProductRecipeMemory, Array based on Current Station No, the read out from fbGnrProductRecipeMemory is based on this Product Recipe Step No*)
	DSfbGnrProductRecipeMemoryOut 		: DS_fbGnrProductRecipeMemoryOut;						(* Input - Link with fbGnrProductRecipeMemory, all the read out info from fbGnrProductRecipeMemory will store in this DataStucture*)

	ARbArmReady							: ARRAY [1..iArmQty] OF BOOL;								(* Input - From ArmPnpFB, This signal is used to confirm if the arm is ready and idling*)
	ARiStnNoToCalledArm					: ARRAY [0..iArmQty] OF INT; 									(* Output - Link with fbArmPnP, Array based on Arm No, The Int will store which Station that calling the Arm*)
	ARDSGnrFeedArmPnpParameter		: ARRAY [0..iArmQty] OF DSGnr_CalledArmPnpParameter; 	(* Output - Link with fbArmPnP, Array based on Current Station No, Arm should move based on this DataStructure Info*)

	DSLdBasketInfo		 				: DS_BasketInfo;									(*Input - Loading CONFIRM Basket Info*)
	DSUldBasketInfo		 				: DS_BasketInfo;									(*Input - Uloading CONFIRM Basket Info*)
	ARDsStnBasketInfo					: ARRAY [1..iStnQty] OF DS_BasketInfo;				(*Input - Station Basket Info*)


END_VAR

VAR_OUTPUT PERSISTENT

	DSGnrBufferCalledArmPnpParameter 	: DSGnr_CalledArmPnpParameter;							(* Internal used, Buffer Data Structure read out from fbGnrProductRecipeMemory*)
	DSGnrBuffersPnpSequenceDescription	: STRING (99);													(* Internal used, Buffer Description read out from fbGnrProductRecipeMemory*)
	ARiPreviousStnSeqTotalProcessTime 	: ARRAY [0..iProductRecipeArrayQty] OF INT;				(* Internal used, Previous Total Process Time will save into this Array, Array based on StationSequenceNo*)
	iCallStep									: INT;															(* Internal used, to monitor the current Step so that you can indentify the error of this function block if stucked*)

END_VAR
VAR PERSISTENT
	bBasketDetectedRE						: R_TRIG;
	iCallCheck								: INT;
	bArmPnpSequenceCallEn				: BOOL;
	bStnSeqProcessCompletedRE			: R_TRIG;
	iCallArmCountDownTime				: INT;
	bCallArmEnInt								: BOOL;


END_VAR
VAR
	bBasketDetectedFE						: F_TRIG;
	bCallProductRecipeStorageEn			: BOOL;
	bTestCallArm								: BOOL;

	DSCurrentStationBasketInfo: DS_BasketInfo;
	DSEmptyBasketInfo: DS_BasketInfo;
	bPickStationBasketAvailable: BOOL;
	bTransferStationBasketAvailable: BOOL;
	bTransferStationBasketNotAvailable: BOOL;
	iCurrentStationAddressInt: INT;
	iTrackerCallArmCountDownTime: INT;
(*	bAlternateStnEnableFound: BOOL;*)
(*	iCheckAlternateStnEnFL: INT;*)
	bPickAltStnIDFound: BOOL;
	iPickAlternateStnFindFL: INT;
	iPickAlternateSetFindFL: INT;
	iPickAltStnTransferFL : INT;
	ARiBufferPickAltStn: ARRAY [1..iAlternateStnQty] OF INT;

	bTransferAltStnIDFound: BOOL;
	iTransferAlternateStnFindFL: INT;
	iTransferAlternateSetFindFL: INT;
	iTransferAltStnTransferFL : INT;
	ARiBufferTransferAltStn: ARRAY [1..iAlternateStnQty] OF INT;

	iCheckTrfStnBktFL: INT;
	iTransferStnNo: INT;
	iAltTransferStnNo: INT;
END_VAR

(*Check if Loading Stn Detected, Switch the CurrentStatonAddress to 0*)
IF iLdStnID = iCurrentStationAddress THEN
iCurrentStationAddressInt := 0;
ELSE
iCurrentStationAddressInt := iCurrentStationAddress;
END_IF


(*Check if Alternate Stn Matched with Current (Pick) Station*)
bPickAltStnIDFound := FALSE;
iPickAlternateSetFindFL := 1;
	FOR iPickAlternateSetFindFL := 1 TO iAlternateSetQty DO
		IF iPickAlternateSetFindFL >= 1 AND iPickAlternateSetFindFL <= iAlternateSetQty THEN
			IF ARbAlternateStnEn[iPickAlternateSetFindFL] THEN
			iPickAlternateStnFindFL := 1; (*Find Stn ID matching*)
				FOR iPickAlternateStnFindFL := 1 TO iAlternateStnQty DO
					IF iPickAlternateStnFindFL >= 1 AND iPickAlternateStnFindFL <= iAlternateStnQty THEN
						IF iCurrentStationAddress = AR2SiAlternateStn[iPickAlternateSetFindFL , iPickAlternateStnFindFL] THEN
							bPickAltStnIDFound := TRUE;
							iPickAltStnTransferFL := 1;
								FOR iPickAltStnTransferFL := 1 TO iAlternateStnQty DO
									IF iPickAltStnTransferFL >= 1 AND iPickAltStnTransferFL <= iAlternateStnQty THEN
										ARiBufferPickAltStn[iPickAltStnTransferFL] := AR2SiAlternateStn[iPickAlternateSetFindFL , iPickAltStnTransferFL];
									END_IF
								END_FOR
							iPickAlternateSetFindFL := iAlternateSetQty+1;
							iPickAlternateStnFindFL := iAlternateStnQty+1;
							iPickAltStnTransferFL := iAlternateStnQty+1;

						END_IF
					END_IF
				END_FOR
			END_IF
		END_IF
	END_FOR

(*Check if Alternate Stn Matched with Transfer Station*)

bTransferAltStnIDFound := FALSE;
IF iCallStep = 3 THEN
iTransferAlternateSetFindFL := 1;
	FOR iTransferAlternateSetFindFL := 1 TO iAlternateSetQty DO
		IF iTransferAlternateSetFindFL >= 1 AND iTransferAlternateSetFindFL <= iAlternateSetQty THEN
			IF ARbAlternateStnEn[iTransferAlternateSetFindFL] THEN
			iTransferAlternateStnFindFL := 1; (*Find Stn ID matching*)
				FOR iTransferAlternateStnFindFL := 1 TO iAlternateStnQty DO
					IF iTransferAlternateStnFindFL >= 1 AND iTransferAlternateStnFindFL <= iAlternateStnQty THEN
						IF DSGnrBufferCalledArmPnpParameter.iTransferStationNo = AR2SiAlternateStn[iTransferAlternateSetFindFL , iTransferAlternateStnFindFL] THEN
							bTransferAltStnIDFound := TRUE;
							iTransferAltStnTransferFL := 1;
								FOR iTransferAltStnTransferFL := 1 TO iAlternateStnQty DO
									IF iTransferAltStnTransferFL >= 1 AND iTransferAltStnTransferFL <= iAlternateStnQty THEN
										ARiBufferTransferAltStn[iTransferAltStnTransferFL] := AR2SiAlternateStn[iTransferAlternateSetFindFL , iTransferAltStnTransferFL];
									END_IF
								END_FOR
							iTransferAlternateSetFindFL := iAlternateSetQty+1;
							iTransferAlternateStnFindFL := iAlternateStnQty+1;
							iTransferAltStnTransferFL := iAlternateStnQty+1;

						END_IF
					END_IF
				END_FOR
			END_IF
		END_IF
	END_FOR
END_IF
(*Define Current Station Basket Info*)
IF iCurrentStationAddress = iLdStnID THEN
DSCurrentStationBasketInfo := DSLdBasketInfo;
ELSIF iCurrentStationAddress = iUldStnID THEN
DSCurrentStationBasketInfo := DSUldBasketInfo;
ELSIF iCurrentStationAddress >= 1 AND iCurrentStationAddress <= iStnQty THEN
DSCurrentStationBasketInfo := ARDsStnBasketInfo[iCurrentStationAddress];
ELSE
DSCurrentStationBasketInfo := DSEmptyBasketInfo;
END_IF


(* Check if no one called Data From DSfbGnrProductRecipeMemory *)
iCallCheck := 1;
FOR iCallCheck := 1 TO iStnQty DO
		IF ARbProductRecipeCallEn[iCallCheck] THEN
		bArmPnpSequenceCallEn := TRUE;
		iCallCheck := 90;
		END_IF
END_FOR

IF iCallCheck > iStnQty AND iCallCheck <= (iStnQty+2) THEN
bArmPnpSequenceCallEn := FALSE;
END_IF


(*[][][][][][][][][][][][][][][][][][][][][][][][][][][][][][][][][][][][][][][][][][][][][][][][][][][][][][][][][][][][][][][][][][][][][][][][][][][][][][][][][][][][][][][][][][][][][][][][][][][]*)
(*Store Previous Total Process Time by Program No*)
bStnSeqProcessCompletedRE(CLK:=bStnSeqProcessCompleted , Q=> );

IF bStnSeqProcessCompletedRE.Q AND (*ARiPreviousStnSeqTotalProcessTime[*)DSCurrentStationBasketInfo.iStationSeqenceRecipeNo(*]*) > 0 AND (*ARiPreviousStnSeqTotalProcessTime[*)DSCurrentStationBasketInfo.iStationSeqenceRecipeNo(*]*) <= iProductRecipeArrayQty THEN
ARiPreviousStnSeqTotalProcessTime[DSCurrentStationBasketInfo.iStationSeqenceRecipeNo] := iPreviousStnSeqProcessTotalTime ;
END_IF


(*[][][][][][][][][][][][][][][][][][][][][][][][][][][][][][][][][][][][][][][][][][][][][][][][][][][][][][][][][][][][][][][][][][][][][][][][][][][][][][][][][][][][][][][][][][][][][][][][][][][]*)
(*Call Arm Activation*)

IF (*NOT DSStnSeqProOutput.b12SlowPull AND*) bStnSeqProcessInProgressFlag OR bStnSeqProcessCompleted THEN
	iCallArmCountDownTime := ARiPreviousStnSeqTotalProcessTime[DSCurrentStationBasketInfo.iStationSeqenceRecipeNo] - iCurrentStnSeqProcessTotalTime;
END_IF
(*
IF DSStnSeqProOutput.b12SlowPull AND bStnSeqProcessInProgressFlag OR bStnSeqProcessCompleted THEN
	iCallArmCountDownTime := iTotalProcessTimeSV - iCurrentStnSeqProcessTotalTime;
END_IF
*)

iTrackerCallArmCountDownTime := iTotalProcessTimeSV - iCurrentStnSeqProcessTotalTime;

IF
(iCurrentStationAddress <> iLdStnID AND NOT bTrackerEN  AND iCurrentStnSeqProcessTotalTime > 0 AND iCallArmCountDownTime >= 0 AND iCallArmCountDownTime <= iPreCallArmTime AND bStnSeqProcessInProgressFlag)
OR
(iCurrentStationAddress <> iLdStnID AND bTrackerEN AND bTrackerBasedOnPreviousTime  AND iCurrentStnSeqProcessTotalTime > 0 AND iCallArmCountDownTime >= 0 AND iCallArmCountDownTime <= iPreCallArmTime AND bStnSeqProcessInProgressFlag)
OR
(iCurrentStationAddress <> iLdStnID AND bTrackerEN AND NOT bTrackerBasedOnPreviousTime AND iCurrentStnSeqProcessTotalTime > 0 AND iTrackerCallArmCountDownTime >= 0 AND iTrackerCallArmCountDownTime <= iPreCallArmTime AND bStnSeqProcessInProgressFlag)
OR
bStnSeqProcessCompleted
OR
bTestCallArm
THEN
bCallArmEnInt := TRUE;
ELSE
bCallArmEnInt := FALSE;
END_IF

(*Check PickStation Basket Availability *)
IF (*DSGnrBufferCalledArmPnpParameter.iPickStationNo*)iCurrentStationAddress = iLdStnID AND DSLdBasketInfo.bAvailibility THEN
bPickStationBasketAvailable := TRUE;
ELSIF (*DSGnrBufferCalledArmPnpParameter.iPickStationNo*)iCurrentStationAddress = iUldStnID AND DSUldBasketInfo.bAvailibility THEN
bPickStationBasketAvailable := TRUE;
ELSIF (*DSGnrBufferCalledArmPnpParameter.iPickStationNo*)iCurrentStationAddress >= 1 AND  (*DSGnrBufferCalledArmPnpParameter.iPickStationNo*)iCurrentStationAddress <= iStnQty AND ARDsStnBasketInfo[(*DSGnrBufferCalledArmPnpParameter.iPickStationNo*)iCurrentStationAddress].bAvailibility THEN
bPickStationBasketAvailable := TRUE;
ELSE
bPickStationBasketAvailable := FALSE;
END_IF
(*
(*Check TransferStation Basket Availability *)
IF DSGnrBufferCalledArmPnpParameter.iTransferStationNo = iLdStnID AND DSLdBasketInfo.bAvailibility THEN
bTransferStationBasketAvailable := TRUE;
ELSIF DSGnrBufferCalledArmPnpParameter.iTransferStationNo = iUldStnID AND DSUldBasketInfo.bAvailibility THEN
bTransferStationBasketAvailable := TRUE;
ELSIF DSGnrBufferCalledArmPnpParameter.iTransferStationNo >= 1 AND  DSGnrBufferCalledArmPnpParameter.iTransferStationNo <= iStnQty AND ARDsStnBasketInfo[DSGnrBufferCalledArmPnpParameter.iTransferStationNo].bAvailibility THEN
bTransferStationBasketAvailable := TRUE;
ELSE
bTransferStationBasketAvailable := FALSE;
END_IF
*)

IF bTransferAltStnIDFound THEN
	iCheckTrfStnBktFL := 1;
	bTransferStationBasketAvailable := TRUE;
	iAltTransferStnNo := 0;
	FOR iCheckTrfStnBktFL := 1 TO iAlternateStnQty DO
	
		IF iCheckTrfStnBktFL >= 1 AND iCheckTrfStnBktFL <= iAlternateStnQty THEN

			IF ARiBufferTransferAltStn[iCheckTrfStnBktFL] = iLdStnID AND NOT DSLdBasketInfo.bAvailibility THEN
			bTransferStationBasketAvailable := FALSE;
			iAltTransferStnNo := ARiBufferTransferAltStn[iCheckTrfStnBktFL];
			iCheckTrfStnBktFL := iAlternateStnQty+1;

			ELSIF ARiBufferTransferAltStn[iCheckTrfStnBktFL] = iUldStnID AND NOT DSUldBasketInfo.bAvailibility THEN
			bTransferStationBasketAvailable := FALSE;
			iAltTransferStnNo := ARiBufferTransferAltStn[iCheckTrfStnBktFL];
			iCheckTrfStnBktFL := iAlternateStnQty+1;

			ELSIF ARiBufferTransferAltStn[iCheckTrfStnBktFL] >= 1 AND ARiBufferTransferAltStn[iCheckTrfStnBktFL] <= iStnQty AND NOT  ARDsStnBasketInfo[ARiBufferTransferAltStn[iCheckTrfStnBktFL]].bAvailibility THEN
			bTransferStationBasketAvailable := FALSE;
			iAltTransferStnNo := ARiBufferTransferAltStn[iCheckTrfStnBktFL];
			iCheckTrfStnBktFL := iAlternateStnQty+1;

			END_IF
	
		END_IF

	END_FOR

ELSE

	IF DSGnrBufferCalledArmPnpParameter.iTransferStationNo = iLdStnID AND DSLdBasketInfo.bAvailibility THEN
	bTransferStationBasketAvailable := TRUE;
	ELSIF DSGnrBufferCalledArmPnpParameter.iTransferStationNo = iUldStnID AND DSUldBasketInfo.bAvailibility THEN
	bTransferStationBasketAvailable := TRUE;
	ELSIF DSGnrBufferCalledArmPnpParameter.iTransferStationNo >= 1 AND  DSGnrBufferCalledArmPnpParameter.iTransferStationNo <= iStnQty AND ARDsStnBasketInfo[DSGnrBufferCalledArmPnpParameter.iTransferStationNo].bAvailibility THEN
	bTransferStationBasketAvailable := TRUE;
	ELSE
	bTransferStationBasketAvailable := FALSE;
	END_IF
	
END_IF

IF bCallArmEnInt
AND bPickStationBasketAvailable
AND NOT bTransferStationBasketAvailable
AND ARbArmReady[DSGnrBufferCalledArmPnpParameter.iCallArmNo]
AND  ARiStnNoToCalledArm[DSGnrBufferCalledArmPnpParameter.iCallArmNo] = 0
AND iCallStep = 3
THEN

	IF bTransferAltStnIDFound THEN
		ARDSGnrFeedArmPnpParameter[DSGnrBufferCalledArmPnpParameter.iCallArmNo] := DSGnrBufferCalledArmPnpParameter;
		ARDSGnrFeedArmPnpParameter[DSGnrBufferCalledArmPnpParameter.iCallArmNo].iPickStationNo := iCurrentStationAddress;
		ARDSGnrFeedArmPnpParameter[DSGnrBufferCalledArmPnpParameter.iCallArmNo].iTransferStationNo := iAltTransferStnNo;

		ARiStnNoToCalledArm[DSGnrBufferCalledArmPnpParameter.iCallArmNo]  := iCurrentStationAddress;

	ELSE

		ARDSGnrFeedArmPnpParameter[DSGnrBufferCalledArmPnpParameter.iCallArmNo] := DSGnrBufferCalledArmPnpParameter;
		ARDSGnrFeedArmPnpParameter[DSGnrBufferCalledArmPnpParameter.iCallArmNo].iPickStationNo := iCurrentStationAddress;
		ARiStnNoToCalledArm[DSGnrBufferCalledArmPnpParameter.iCallArmNo]  := iCurrentStationAddress;

	END_IF

END_IF




(*[][][][][][][][][][][][][][][][][][][][][][][][][][][][][][][][][][][][][][][][][][][][][][][][][][][][][][][][][][][][][][][][][][][][][][][][][][][][][][][][][][][][][][][][][][][][][][][][][][][]*)
(*Start Call *)
IF bBasketDetectedFE.Q THEN
iCallStep := 0;
END_IF

bBasketDetectedRE(CLK:=DSCurrentStationBasketInfo.bAvailibility , Q=> );
bBasketDetectedFE(CLK:=DSCurrentStationBasketInfo.bAvailibility , Q=> );
(*
IF bBasketDetectedRE.Q THEN
DSCurrentStationBasketInfo.iStationSeqenceRecipeNo :=  0;
END_IF
*)
IF DSCurrentStationBasketInfo.bAvailibility AND NOT bCallProductRecipeStorageEn AND NOT bArmPnpSequenceCallEn THEN
ARbProductRecipeCallEn[iCurrentStationAddressInt] := TRUE;
iCallStep := 1;
bCallProductRecipeStorageEn := TRUE;
END_IF

IF DSCurrentStationBasketInfo.bAvailibility AND DSCurrentStationBasketInfo.iStationSeqenceRecipeNo > 0 THEN (*New, Make sure during ArmPnP, must write the StnSeqRecipeNo to BasketInfo before put the basket to station*)
bStnSeqProcessSt := TRUE;
ELSE
bStnSeqProcessSt := FALSE;
END_IF


CASE iCallStep OF

0:
ARbProductRecipeCallEn[iCurrentStationAddressInt] := FALSE;
bCallProductRecipeStorageEn := FALSE;
bStnSeqProcessSt := FALSE;


1:

ARiProductRecipeNoCall[iCurrentStationAddressInt] := DSCurrentStationBasketInfo.iProductRecipeNo;
ARiProductRecipeStepCall[iCurrentStationAddressInt] := DSCurrentStationBasketInfo.iProductRecipeStepNo+1(*New*);
ARbProductRecipeCallEn[iCurrentStationAddressInt] := TRUE;
iCallStep := 2;

2:

IF DSfbGnrProductRecipeMemoryOut.bCallCompleted
AND  DSfbGnrProductRecipeMemoryOut.iCalledProductRecipeNo = DSCurrentStationBasketInfo.iProductRecipeNo
AND DSfbGnrProductRecipeMemoryOut.iCalledProductRecipeStep = DSCurrentStationBasketInfo.iProductRecipeStepNo+1(*New*)
AND NOT DSfbGnrProductRecipeMemoryOut.bCallPickStationNoErr
AND NOT DSfbGnrProductRecipeMemoryOut.bCallTransferStationNoErr
AND NOT DSfbGnrProductRecipeMemoryOut.bCallUpDownPatternMemoryErr
AND NOT DSfbGnrProductRecipeMemoryOut.bInvalidProductRecipeNoErrHold
AND NOT DSfbGnrProductRecipeMemoryOut.bInvalidProductRecipeNoErrPulse
AND NOT DSfbGnrProductRecipeMemoryOut.bInvalidProductRecipeStepErrHold
AND NOT DSfbGnrProductRecipeMemoryOut.bInvalidProductRecipeStepErrPulse
THEN

DSGnrBufferCalledArmPnpParameter := DSfbGnrProductRecipeMemoryOut.DSGnrCalledArmPnpParameter;
DSGnrBuffersPnpSequenceDescription := DSfbGnrProductRecipeMemoryOut.sProductRecipeDescription;
(*DSCurrentStationBasketInfo.iStationSeqenceRecipeNo := DSGnrBufferCalledArmPnpParameter.iStnSeqRecipeNo;*) (*New*)
ARbProductRecipeCallEn[iCurrentStationAddressInt] := FALSE;
iCallStep := 3;
END_IF

IF DSfbGnrProductRecipeMemoryOut.bCallCompleted
AND (  DSfbGnrProductRecipeMemoryOut.iCalledProductRecipeNo <> DSCurrentStationBasketInfo.iProductRecipeNo
OR DSfbGnrProductRecipeMemoryOut.iCalledProductRecipeStep <> DSCurrentStationBasketInfo.iProductRecipeStepNo+1(*New*))
THEN
ARbProductRecipeCallEn[iCurrentStationAddressInt] := FALSE;
iCallStep := 11;
END_IF


IF DSfbGnrProductRecipeMemoryOut.bCallCompleted
AND (DSfbGnrProductRecipeMemoryOut.bCallPickStationNoErr
OR DSfbGnrProductRecipeMemoryOut.bCallTransferStationNoErr
OR DSfbGnrProductRecipeMemoryOut.bCallUpDownPatternMemoryErr
OR DSfbGnrProductRecipeMemoryOut.bInvalidProductRecipeNoErrHold
OR DSfbGnrProductRecipeMemoryOut.bInvalidProductRecipeNoErrPulse
OR DSfbGnrProductRecipeMemoryOut.bInvalidProductRecipeStepErrHold
OR DSfbGnrProductRecipeMemoryOut.bInvalidProductRecipeStepErrPulse)
THEN
ARbProductRecipeCallEn[iCurrentStationAddressInt] := FALSE;
iCallStep := 12;
END_IF

3: (*Complete without Error*);
ARbProductRecipeCallEn[iCurrentStationAddressInt] := FALSE;


11: (*Program No or Step No Not Matching*);

12: (*Error when call data *);

END_CASE


(*[][][][][][][][][][][][][][][][][][][][][][][][][][][][][][][][][][][][][][][][][][][][][][][][][][][][][][][][][][][][][][][][][][][][][][][][][][][][][][][][][][][][][][][][][][][][][][][][][][][]*)

END_FUNCTION_BLOCK

// ---- FBs/B_JKS_NewFB/FBP-Memory_Sub/fbSingleArmBasketMemoryV2.TcPOU
FUNCTION_BLOCK fbSingleArmBasketMemoryV2
VAR_INPUT

	iCurStationNo : INT;
	bConfirmCondition : BOOL;
	bConfirmTrigger : BOOL;
	bTransferCondition : BOOL;
	bTransferTrigger : BOOL;


END_VAR


VAR_OUTPUT



END_VAR

VAR

	bConfirmTriggerDIFU : R_TRIG;
	TransferTriggerDIFU : R_TRIG;
	EmptyDsBasketInfo : DS_BasketInfo;
	iCTCompareResult: DINT;
	iTTCompareResult: DINT;
	bConfirmTriggerHR: BOOL;
	tConfirmTriggerDoff: TON;
	tTransferTriggerDoff: TON;
	bTransferTriggerHR: BOOL;
END_VAR

VAR_IN_OUT
	DSPreTransBasketInfo : DS_BasketInfo;
	DSCurConfirmBasketInfo : DS_BasketInfo;
	DSCurTransBasketInfo : DS_BasketInfo;

(*
	bPreTransBasket : BOOL;
	bCurConfirmBasket : BOOL;
	bCurTransBasket : BOOL;

	sPreTransStringMemory1 : STRING(50);
	sPreTransStringMemory2 : STRING(50);
	sPreTransStringMemory3 : STRING(50);
	sPreTransStringMemory4 : STRING(50);
	sPreTransStringMemory5 : STRING(50);
	sPreTransStringMemory6 : STRING(50);
	iPreTransRecipeNo : INT;
	iPrePickedBasketStationNo : INT;

	sCurConfirmStringMemory1 : STRING(50);
	sCurConfirmStringMemory2 : STRING(50);
	sCurConfirmStringMemory3 : STRING(50);
	sCurConfirmStringMemory4 : STRING(50);
	sCurConfirmStringMemory5 : STRING(50);
	sCurConfirmStringMemory6 : STRING(50);
	iCurConfirmRecipeNo : INT;



	sCurTransStringMemory1 : STRING(50);
	sCurTransStringMemory2 : STRING(50);
	sCurTransStringMemory3 : STRING(50);
	sCurTransStringMemory4 : STRING(50);
	sCurTransStringMemory5 : STRING(50);
	sCurTransStringMemory6 : STRING(50);
	iCurTransRecipeNo : INT;
	iCurPickedBasketStationNo : INT;

*)
END_VAR

(*Generate Basket Confirm Bit *)

IF DSPreTransBasketInfo.iProductRecipeNo <> 0 THEN
DSPreTransBasketInfo.bAvailibility := TRUE;
ELSE
DSPreTransBasketInfo.bAvailibility := FALSE;
END_IF

IF DSCurConfirmBasketInfo.iProductRecipeNo <> 0 THEN
DSCurConfirmBasketInfo.bAvailibility := TRUE;
ELSE
DSCurConfirmBasketInfo.bAvailibility := FALSE;
END_IF

IF DSCurTransBasketInfo.iProductRecipeNo <> 0 THEN
DSCurTransBasketInfo.bAvailibility := TRUE;
ELSE
DSCurTransBasketInfo.bAvailibility := FALSE;
END_IF


(* PreTrans -> CurConfirm *)
bConfirmTriggerDIFU(CLK:=bConfirmTrigger , Q=> );
tConfirmTriggerDoff(IN:=bConfirmTriggerHR , PT:=t#1s , Q=> , ET=> );


IF tConfirmTriggerDoff.Q THEN
bConfirmTriggerHR := FALSE;
END_IF


IF bConfirmTriggerDIFU.Q THEN
bConfirmTriggerHR := TRUE;
END_IF


IF (*bConfirmTriggerHR*)bConfirmTriggerDIFU.Q AND bConfirmCondition THEN

	IF DSPreTransBasketInfo.iProductRecipeNo <> 0 AND DSCurConfirmBasketInfo.iProductRecipeNo = 0 THEN

			DSCurConfirmBasketInfo := DSPreTransBasketInfo;

			iCTCompareResult := MEMCMP(ADR(DSCurConfirmBasketInfo), ADR(DSPreTransBasketInfo), SIZEOF(DSPreTransBasketInfo));

			IF iCTCompareResult = 0 THEN
			DSPreTransBasketInfo := EmptyDsBasketInfo;
			DSCurConfirmBasketInfo.iCurrentStationNo := iCurStationNo;
			END_IF


			IF DSCurConfirmBasketInfo.iProductRecipeNo <> 0 THEN
			DSCurConfirmBasketInfo.iPreviousStationNo := 0;
			END_IF

	END_IF

END_IF

(* CurConfirm -> CurTransfer *)
TransferTriggerDIFU(CLK:=bTransferTrigger , Q=> );

tTransferTriggerDoff(IN:=bTransferTriggerHR , PT:=t#1s , Q=> , ET=> );


IF tTransferTriggerDoff.Q THEN
bTransferTriggerHR := FALSE;
END_IF


IF TransferTriggerDIFU.Q THEN
bTransferTriggerHR := TRUE;
END_IF



IF (*bTransferTriggerHR*)TransferTriggerDIFU.Q AND bTransferCondition THEN


	IF DSCurConfirmBasketInfo.iProductRecipeNo <> 0 AND DSCurTransBasketInfo.iProductRecipeNo = 0 THEN
			DSCurTransBasketInfo := DSCurConfirmBasketInfo;

			iTTCompareResult := MEMCMP(ADR(DSCurTransBasketInfo), ADR(DSCurConfirmBasketInfo), SIZEOF(DSCurConfirmBasketInfo));

			IF iTTCompareResult = 0 THEN
			DSCurConfirmBasketInfo := EmptyDsBasketInfo;
			DSCurTransBasketInfo.iPreviousStationNo := iCurStationNo;
			END_IF


			IF DSCurTransBasketInfo.iProductRecipeNo <> 0 THEN
			DSCurTransBasketInfo.iCurrentStationNo := 0;
			END_IF

	END_IF


END_IF

END_FUNCTION_BLOCK

// ---- FBs/B_JKS_NewFB/FBP-Memory_Sub/fbStationSequenceRecipe.TcPOU
FUNCTION_BLOCK fbStationSequenceRecipe

VAR_INPUT
	bSavePB : BOOL;
	bLoadPB : BOOL;
	bCopyPB : BOOL;
(*	iCopyFromSubRecipeNo : INT;*)
	iCopyToSubRecipeNo : INT;
END_VAR


VAR_IN_OUT PERSISTENT

	iStationSequenceRecipeNo: INT; (* 10 sets of Station Sequence Recipe *)
	sStationSequenceRecipeDescription : STRING(50); (* Description of Station Sequence Recipe - Naming*)
	DsInStationSequenceRecipeMemory : DS_StationSequenceRecipeMemory;
(*	AR10iStationSubProNo : ARRAY [0..10] OF INT; (* 10 units of SubProcessProgramNo / Steps *)
	AR10iCycle : ARRAY [0..10] OF INT; (* 10 units of Integer to Store the Cycle needed on the specified Steps. at least "1" *)
	AR10iRepeatFromStepNo : ARRAY [0..10] OF INT; (* 10 units of Integer to when Cycle repeat, it will repeat from Which Steps  *)
*)




	Call_iStationSequenceRecipe : INT;
	bCallPB: BOOL;
(*	bCallPBEnable : BOOL;*)
(*	ScrMapCall_iStationSequenceRecipe : INT;*)




END_VAR
VAR_OUTPUT
	bSaveInd: BOOL;
	bLoadInd: BOOL;
	bCallCompleted : BOOL;
	bInvalidCallStationSequenceNoHold: BOOL;
	bInvalidCallStationSequenceNoPulse: BOOL;
(*	bInvalidScrMapCallStationSequenceNo : BOOL;*)
	Call_sSequenceRecipeDescription : STRING(50);
	Call_DsStationSequenceRecipeMemory : DS_StationSequenceRecipeMemory;

(*	Call_AR10iStationSubProNo : ARRAY [0..10] OF INT;
	Call_AR10iCycle : ARRAY [0..10] OF INT;
	Call_AR10iRepeatFromStepNo : ARRAY [0..10] OF INT;
*)
(*	ScrMapCall_sSequenceRecipeDescription : STRING(50);
	ScrMapCall_AR10iStationSubProNo : ARRAY [0..10] OF INT;
	ScrMapCall_AR10iCycle : ARRAY [0..10] OF INT;
	ScrMapCall_AR10iRepeatFromStepNo : ARRAY [0..10] OF INT;*)





END_VAR
VAR
	SaveIndHr: BOOL;
	LoadIndHr: BOOL;

	SaveTimerDelay: TON;
	LoadTimerDelay: TON;
	SelfCheckTimer: TON;
	bLoadEn: BOOL;
	SelfCheckloopSequenceRecipe: BOOL;
	PreviousNoSequenceRecipe: INT;

	LoadDF : R_TRIG;
	LoadENDF : R_TRIG;

	SaveDF: R_TRIG;
	CallIntervalTimer: TON;
	CallIntervalDIFU: R_TRIG;

	bCallCompletedHR: BOOL;
	bCallCompletedHRRE: R_TRIG;
	CallCompletedTimer: TON;
	CallSelfCheckTimer : TON;
	CallSelfCheckloop : BOOL;

	CallSelfCheckRE: R_TRIG;
	CallStep: INT;
	CallSelfCheckHR: BOOL;
	bCallPBRE: R_TRIG;

	LoadFL: INT;
	SaveFL: INT;
	PreviousStationRequenceRecipeCallNo: INT;
	CallSFL: INT;
	febInvalidCallStationSequenceNo: F_TRIG;



	rebInvalidCallStationSequenceNo: R_TRIG;
	tInvalidCallStationSequenceNoPulseTimer: TON;
	CopyDF: R_TRIG;
END_VAR

VAR PERSISTENT

	ARDsStorageStationSequenceRecipeMemory : ARRAY [1..iStationSequenceRecipeArrayQty] OF DS_StationSequenceRecipeMemory;
	ARsStorageStationSequenceRecipeDescription: ARRAY [0..iStationSequenceRecipeArrayQty] OF STRING(50);


END_VAR

IF iStationSequenceRecipeNo < 1 THEN
iStationSequenceRecipeNo := 1;
END_IF

IF iStationSequenceRecipeNo > iStationSequenceRecipeArrayQty THEN
iStationSequenceRecipeNo := iStationSequenceRecipeArrayQty;
END_IF

(*Add New*)
ARsStorageStationSequenceRecipeDescription[0] := '- - - End Step - - -';


(*Load and Save Indicator*)
IF bSavePB THEN
SaveIndHr := TRUE;
END_IF

SaveTimerDelay(IN:=SaveIndHr, PT := T#1s, Q=>, ET=>);
IF SaveTimerDelay.Q THEN
SaveIndHr := FALSE;
END_IF

IF SaveIndHr AND NOT SaveTimerDelay.Q THEN
bSaveInd := TRUE;
ELSE
bSaveInd := FALSE;
END_IF

IF bLoadPB THEN
LoadIndHr := TRUE;
END_IF

LoadTimerDelay(IN:=LoadIndHr, PT := T#1s, Q=>, ET=>);
IF loadtimerdelay.Q THEN
LoadIndHr := FALSE;
END_IF

IF loadIndHr AND NOT LoadTimerDelay.Q THEN
bLoadInd := TRUE;
ELSE
bLoadInd := FALSE;
END_IF

IF iStationSequenceRecipeNo <> PreviousNoSequenceRecipe THEN
bLoadEn := TRUE;
ELSE
bLoadEn := FALSE;
END_IF


(* Load Recipe *)

LoadDF(CLK:=bLoadPB,Q=>);
LoadENDF(CLK:=bLoadEn,Q=>);

IF LoadDF.Q OR LoadENDF.Q THEN

DsInStationSequenceRecipeMemory := ARDsStorageStationSequenceRecipeMemory[iStationSequenceRecipeNo];
sStationSequenceRecipeDescription := ARsStorageStationSequenceRecipeDescription[iStationSequenceRecipeNo];
PreviousNoSequenceRecipe := iStationSequenceRecipeNo  ;

END_IF


(* Save Recipe *)

SaveDF(CLK:=bSavePB,Q=>);

IF SaveDF.Q THEN

ARDsStorageStationSequenceRecipeMemory[iStationSequenceRecipeNo] := DsInStationSequenceRecipeMemory;
ARsStorageStationSequenceRecipeDescription[iStationSequenceRecipeNo] := sStationSequenceRecipeDescription;

END_IF


(*Copy Recipe*)

CopyDF(CLK:=bCopyPB,Q=>);

IF CopyDF.Q THEN

ARDsStorageStationSequenceRecipeMemory[iCopyToSubRecipeNo] := ARDsStorageStationSequenceRecipeMemory[iStationSequenceRecipeNo];
ARsStorageStationSequenceRecipeDescription[iCopyToSubRecipeNo] := ARsStorageStationSequenceRecipeDescription[iStationSequenceRecipeNo];

END_IF




(* Call Recipe *)
(* ---- Call Recipe Complete Flag ---*)

(*
CallCompletedTimer(IN:=bCallCompleted , PT:=t#0.5s , Q=> , ET=> );
*)
IF (*CallCompletedTimer.Q*) NOT bCallPB THEN
bCallCompleted := FALSE;
END_IF
(*
CallSelfCheckRE(CLK:=PreviousStationRequenceRecipeCallNo <> Call_iStationSequenceRecipe , Q=> );

IF CallSelfCheckRE.Q THEN
CallSelfCheckHR := TRUE;
END_IF
*)
bCallPBRE(CLK:=bCallPB , Q=> );

IF (Call_iStationSequenceRecipe <= 0 OR Call_iStationSequenceRecipe > iStationSequenceRecipeArrayQty) AND bCallPB THEN
bInvalidCallStationSequenceNoHold := TRUE;
ELSE
bInvalidCallStationSequenceNoHold := FALSE;
END_IF


rebInvalidCallStationSequenceNo(CLK:= bCallPB AND bInvalidCallStationSequenceNoHold  , Q=> );

IF rebInvalidCallStationSequenceNo.Q THEN
bInvalidCallStationSequenceNoPulse := TRUE;
END_IF

tInvalidCallStationSequenceNoPulseTimer(IN:=bInvalidCallStationSequenceNoPulse , PT:=t#0.5s , Q=> , ET=> );

IF tInvalidCallStationSequenceNoPulseTimer.Q OR NOT bCallPB THEN
bInvalidCallStationSequenceNoPulse := FALSE;
END_IF
(*
febInvalidCallStationSequenceNo(CLK:=bInvalidCallStationSequenceNoHold  , Q=> );
*)
IF bCallPBRE.Q AND NOT bInvalidCallStationSequenceNoHold (*OR febInvalidCallStationSequenceNo.Q*) THEN
bCallCompleted := FALSE;
CallStep:= 1;
END_IF


CASE CallStep OF

1:

Call_DsStationSequenceRecipeMemory := ARDsStorageStationSequenceRecipeMemory[Call_iStationSequenceRecipe];
Call_sSequenceRecipeDescription := ARsStorageStationSequenceRecipeDescription[Call_iStationSequenceRecipe];

(*IF NOT bCallPBEnable AND CallSelfCheckHR THEN
CallStep := 10;
ELSIF NOT bCallPBEnable AND NOT CallSelfCheckHR THEN
CallStep := 99;*)


(*IF bCallPBEnable THEN*)
CallStep := 11;


10:
bCallCompleted := TRUE;
CallSelfCheckHR := FALSE;
PreviousStationRequenceRecipeCallNo := Call_iStationSequenceRecipe;
CallStep := 99;

11:

